	REGION D1.6.1
	    //D1.6.1
	    #"D1.6.1"(ConveyorID := _."D1.6.1",
	              ConveyorSensor:=_."ASiGW-MCC001-bw200-C1: Input"."Sensor D1.6.1",
	              Fault := DB_UDI.ProductionLine.Fault.Stop.Conveyor[_."D1.6.1"],
	              Upstream := DB_UDI.ProductionLine.Upstream.Conveyor[_."D1.6.1"],
	              Downstream := DB_UDI.ProductionLine.DownstreamAccu.Stop.Conveyor[_."D1.6.1"],
	              Interlock := DB_UDI.ProductionLine.Interlock.Stop.Conveyor[_."D1.6.1"],
	              RunForward=>_."ASiGW-MCC001-bw200-C1: Output"."Motor D1.6.1",
	              WriteAsiDir=>_."ASiGW-MCC001-bw200-C1: Output"."Dir D1.6.1");
	    
	END_REGION
	
	REGION D1.7.1
	    //D1.7.1
	    #"D1.7.1"(ConveyorID := _."D1.7.1",
	              ConveyorSensor:=_."ASiGW-MCC001-bw200-C1: Input"."Sensor D1.7.10",
	              Fault := DB_UDI.ProductionLine.Fault.Stop.Conveyor[_."D1.7.1"],
	              Upstream := DB_UDI.ProductionLine.Upstream.Conveyor[_."D1.7.1"],
	              Downstream := DB_UDI.ProductionLine.DownstreamAccu.Stop.Conveyor[_."D1.7.1"],
	              Interlock := DB_UDI.ProductionLine.Interlock.Stop.Conveyor[_."D1.7.1"],
	              RunForward=>_."ASiGW-MCC001-bw200-C1: Output"."Motor D1.7.1",
	              WriteAsiDir=>_."ASiGW-MCC001-bw200-C1: Output"."Dir D1.7.1");
	    
	END_REGION
	
	REGION D1.7.2
	    //D1.7.2
	    #"D1.7.2"(ConveyorID := _."D1.7.2",
	              ConveyorSensor:=_."ASiGW-MCC001-bw200-C1: Input"."Sensor D1.7.10",
	              Fault := DB_UDI.ProductionLine.Fault.Stop.Conveyor[_."D1.7.2"],
	              Upstream := DB_UDI.ProductionLine.Upstream.Conveyor[_."D1.7.2"],
	              Downstream := DB_UDI.ProductionLine.DownstreamAccu.Stop.Conveyor[_."D1.7.2"],
	              Interlock := DB_UDI.ProductionLine.Interlock.Stop.Conveyor[_."D1.7.2"],
	              RunForward=>_."ASiGW-MCC001-bw200-C1: Output"."Motor D1.7.2",
	              WriteAsiDir=>_."ASiGW-MCC001-bw200-C1: Output"."Dir D1.7.2");
	    
	END_REGION
	
	REGION D1.7.3
	    //D1.7.3
	    #"D1.7.3"(ConveyorID := _."D1.7.3",
	              ConveyorSensor:=_."ASiGW-MCC001-bw200-C1: Input"."Sensor D1.7.10",
	              Fault := DB_UDI.ProductionLine.Fault.Stop.Conveyor[_."D1.7.3"],
	              Upstream := DB_UDI.ProductionLine.Upstream.Conveyor[_."D1.7.3"],
	              Downstream := DB_UDI.ProductionLine.DownstreamAccu.Stop.Conveyor[_."D1.7.3"],
	              Interlock := DB_UDI.ProductionLine.Interlock.Stop.Conveyor[_."D1.7.3"],
	              RunForward=>_."ASiGW-MCC001-bw200-C1: Output"."Motor D1.7.3",
	              WriteAsiDir=>_."ASiGW-MCC001-bw200-C1: Output"."Dir D1.7.3");
	    
	END_REGION
	
	REGION D1.7.4
	    //D1.7.4
	    #"D1.7.4"(ConveyorID := _."D1.7.4",
	              ConveyorSensor:=_."ASiGW-MCC001-bw200-C1: Input"."Sensor D1.7.10",
	              Fault := DB_UDI.ProductionLine.Fault.Stop.Conveyor[_."D1.7.4"],
	              Upstream := DB_UDI.ProductionLine.Upstream.Conveyor[_."D1.7.4"],
	              Downstream := DB_UDI.ProductionLine.DownstreamAccu.Stop.Conveyor[_."D1.7.4"],
	              Interlock := DB_UDI.ProductionLine.Interlock.Stop.Conveyor[_."D1.7.4"],
	              RunForward=>_."ASiGW-MCC001-bw200-C1: Output"."Motor D1.7.4",
	              WriteAsiDir=>_."ASiGW-MCC001-bw200-C1: Output"."Dir D1.7.4");
	    
	END_REGION
	
	REGION D1.7.5
	    //D1.7.5
	    #"D1.7.5"(ConveyorID := _."D1.7.5",
	              ConveyorSensor:=_."ASiGW-MCC001-bw200-C1: Input"."Sensor D1.7.10",
	              Fault := DB_UDI.ProductionLine.Fault.Stop.Conveyor[_."D1.7.5"],
	              Upstream := DB_UDI.ProductionLine.Upstream.Conveyor[_."D1.7.5"],
	              Downstream := DB_UDI.ProductionLine.DownstreamAccu.Stop.Conveyor[_."D1.7.5"],
	              Interlock := DB_UDI.ProductionLine.Interlock.Stop.Conveyor[_."D1.7.5"],
	              RunForward=>_."ASiGW-MCC001-bw200-C1: Output"."Motor D1.7.5",
	              WriteAsiDir=>_."ASiGW-MCC001-bw200-C1: Output"."Dir D1.7.5");
	    
	END_REGION
	
	REGION D1.7.6
	    //D1.7.6
	    #"D1.7.6"(ConveyorID := _."D1.7.6",
	              ConveyorSensor:=_."ASiGW-MCC001-bw200-C1: Input"."Sensor D1.7.10",
	              Fault := DB_UDI.ProductionLine.Fault.Stop.Conveyor[_."D1.7.6"],
	              Upstream := DB_UDI.ProductionLine.Upstream.Conveyor[_."D1.7.6"],
	              Downstream := DB_UDI.ProductionLine.DownstreamAccu.Stop.Conveyor[_."D1.7.6"],
	              Interlock := DB_UDI.ProductionLine.Interlock.Stop.Conveyor[_."D1.7.6"],
	              RunForward=>_."ASiGW-MCC001-bw200-C1: Output"."Motor D1.7.6",
	              WriteAsiDir=>_."ASiGW-MCC001-bw200-C1: Output"."Dir D1.7.6");
	    
	END_REGION
	
	REGION D1.7.7
	    //D1.7.7
	    #"D1.7.7"(ConveyorID := _."D1.7.7",
	              ConveyorSensor:=_."ASiGW-MCC001-bw200-C1: Input"."Sensor D1.7.10",
	              Fault := DB_UDI.ProductionLine.Fault.Stop.Conveyor[_."D1.7.7"],
	              Upstream := DB_UDI.ProductionLine.Upstream.Conveyor[_."D1.7.7"],
	              Downstream := DB_UDI.ProductionLine.DownstreamAccu.Stop.Conveyor[_."D1.7.7"],
	              Interlock := DB_UDI.ProductionLine.Interlock.Stop.Conveyor[_."D1.7.7"],
	              RunForward => _."ASiGW-MCC001-bw200-C1: Output"."Motor D1.7.7",
	              WriteAsiDir => _."ASiGW-MCC001-bw200-C1: Output"."Dir D1.7.7");
	    
	END_REGION
	
	REGION D1.7.8
	    //D1.7.8
	    #"D1.7.8"(ConveyorID := _."D1.7.8",
	              ConveyorSensor:=_."ASiGW-MCC001-bw200-C1: Input"."Sensor D1.7.10",
	              Fault := DB_UDI.ProductionLine.Fault.Stop.Conveyor[_."D1.7.8"],
	              Upstream := DB_UDI.ProductionLine.Upstream.Conveyor[_."D1.7.8"],
	              Downstream := DB_UDI.ProductionLine.DownstreamAccu.Stop.Conveyor[_."D1.7.8"],
	              Interlock := DB_UDI.ProductionLine.Interlock.Stop.Conveyor[_."D1.7.8"],
	              RunForward=>_."ASiGW-MCC001-bw200-C1: Output"."Motor D1.7.8",
	              WriteAsiDir=>_."ASiGW-MCC001-bw200-C1: Output"."Dir D1.7.8");
	    
	END_REGION
	
	REGION D1.7.9
	    //D1.7.9
	    #"D1.7.9"(ConveyorID := _."D1.7.9",
	              ConveyorSensor:=_."ASiGW-MCC001-bw200-C1: Input"."Sensor D1.7.10",
	               Fault := DB_UDI.ProductionLine.Fault.Stop.Conveyor[_."D1.7.9"],
	               Upstream := DB_UDI.ProductionLine.Upstream.Conveyor[_."D1.7.9"],
	               Downstream := DB_UDI.ProductionLine.DownstreamAccu.Stop.Conveyor[_."D1.7.9"],
	               Interlock := DB_UDI.ProductionLine.Interlock.Stop.Conveyor[_."D1.7.9"],
	               RunForward=>_."ASiGW-MCC001-bw200-C1: Output"."Motor D1.7.9",
	               WriteAsiDir=>_."ASiGW-MCC001-bw200-C1: Output"."Dir D1.7.9");
	     
	END_REGION
	
	REGION D1.7.10
	    //D1.7.10
	    #"D1.7.10"(ConveyorID := _."D1.7.10",
	               ConveyorSensor:=_."ASiGW-MCC001-bw200-C1: Input"."Sensor D1.7.10",
	               Fault := DB_UDI.ProductionLine.Fault.Stop.Conveyor[_."D1.7.10"],
	               Upstream := DB_UDI.ProductionLine.Upstream.Conveyor[_."D1.7.10"],
	               Downstream := DB_UDI.ProductionLine.DownstreamAccu.Stop.Conveyor[_."D1.7.10"],
	               Interlock := DB_UDI.ProductionLine.Interlock.Stop.Conveyor[_."D1.7.10"],
	               RunForward => _."ASiGW-MCC001-bw200-C1: Output"."Motor D1.7.10",
	               WriteAsiDir => _."ASiGW-MCC001-bw200-C1: Output"."Dir D1.7.10");
	    
	END_REGION
	
	REGION D1.8.1
	    //D1.8.1
	    #"D1.8.1"(ConveyorID := _."D1.8.1",
	              ConveyorSensor:=_."ASiGW-MCC001-bw200-C1: Input"."Sensor D1.8.1",
	              Fault := DB_UDI.ProductionLine.Fault.Stop.Conveyor[_."D1.8.1"],
	              Upstream := DB_UDI.ProductionLine.Upstream.Conveyor[_."D1.8.1"],
	              Downstream := DB_UDI.ProductionLine.DownstreamAccu.Stop.Conveyor[_."D1.8.1"],
	              Interlock := DB_UDI.ProductionLine.Interlock.Stop.Conveyor[_."D1.8.1"],
	              RunForward => _."ASiGW-MCC001-bw200-C1: Output"."Motor D1.8.1",
	              WriteAsiDir => _."ASiGW-MCC001-bw200-C1: Output"."Dir D1.8.1");
	    
	END_REGION
	
	REGION D1.8.2
	    //D1.8.2
	    #"D1.8.2"(ConveyorID := _."D1.8.2",
	              ConveyorSensor:=_."ASiGW-MCC001-bw200-C1: Input"."Sensor D1.8.2",
	              Fault := DB_UDI.ProductionLine.Fault.Stop.Conveyor[_."D1.8.2"],
	              Upstream := DB_UDI.ProductionLine.Upstream.Conveyor[_."D1.8.2"],
	              Downstream := DB_UDI.ProductionLine.DownstreamAccu.Stop.Conveyor[_."D1.8.2"],
	              Interlock := DB_UDI.ProductionLine.Interlock.Stop.Conveyor[_."D1.8.2"],
	              RunForward => _."ASiGW-MCC001-bw200-C1: Output"."Motor D1.8.2",
	              WriteAsiDir => _."ASiGW-MCC001-bw200-C1: Output"."Dir D1.8.2");
	    
	END_REGION
	
	REGION D1.8.3
	    //D1.8.3
	    #"D1.8.3"(ConveyorID := _."D1.8.3",
	              ConveyorSensor:=_."ASiGW-MCC001-bw200-C1: Input"."Sensor D1.8.3",
	              Fault := DB_UDI.ProductionLine.Fault.Stop.Conveyor[_."D1.8.3"],
	              Upstream := DB_UDI.ProductionLine.Upstream.Conveyor[_."D1.8.3"],
	              Downstream := DB_UDI.ProductionLine.DownstreamAccu.Stop.Conveyor[_."D1.8.3"],
	              Interlock := DB_UDI.ProductionLine.Interlock.Stop.Conveyor[_."D1.8.3"],
	              RunForward => _."ASiGW-MCC001-bw200-C1: Output"."Motor D1.8.3",
	              WriteAsiDir => _."ASiGW-MCC001-bw200-C1: Output"."Dir D1.8.3");
	    
	END_REGION
	
	REGION D1.9.1 Transfer Unit
	    ////Transfer D1.9.1
	    #"D1.9.2"(TransferID := _."D1.9.1",
	              TransferSensor:=_."ASiGW-MCC001-bw200-C1: Input"."LoadPresence -D1.9.1",
	              Fault := DB_UDI.ProductionLine.Fault.Stop.Conveyor[_."D1.9.1"],
	              Upstream := DB_UDI.ProductionLine.Upstream.Conveyor[_."D1.9.1"],
	              FrontSensor:=_."ASiGW-MCC001-bw200-C1: Input"."FrontSensor -D1.9.1",
	              EndSensor:=_."ASiGW-MCC001-bw200-C1: Input"."EndSensor -D1.9.1",
	              "Left/RightSensor":=_."ASiGW-MCC001-bw200-C1: Input"."LeftSensor -D1.9.1",
	              Downstream := DB_UDI.ProductionLine.DownstreamAccu.Stop.Conveyor[_."D1.9.1"],
	              TransferDirection := DB_ToteTracking.Conveyor[_."D1.9.1"].ToteDir,
	              StartSignal => _."ASiGW-MCC001-bw200-C1: Output"."StartSignal -D1.9.1",
	              Cmd1 =>  _."ASiGW-MCC001-bw200-C1: Output"."Command1 -D1.9.1",
	              Cmd2 => _."ASiGW-MCC001-bw200-C1: Output"."Command2 -D1.9.1",
	              ErrorReset =>  _."ASiGW-MCC001-bw200-C1: Output"."ErrorReset -D1.9.1");
	    
	END_REGION
	
	REGION D1.10.1 Transfer Unit
	    ////Transfer D1.10.1
	    #"D1.10.1"(TransferID := _."D1.10.1",
	              Fault := DB_UDI.ProductionLine.Fault.Stop.Conveyor[_."D1.10.1"],
	              Upstream := DB_UDI.ProductionLine.Upstream.Conveyor[_."D1.10.1"],
	              Downstream := DB_UDI.ProductionLine.DownstreamAccu.Stop.Conveyor[_."D1.10.1"],
	              TransferDirection := DB_ToteTracking.Conveyor[_."D1.10.1"].ToteDir,
	              StartSignal =>  _."ASiGW-MCC001-bw200-C1: Output"."StartSignal -D1.10.1",
	              Cmd1 =>  _."ASiGW-MCC001-bw200-C1: Output"."Command1 -D1.10.1",
	              Cmd2 =>  _."ASiGW-MCC001-bw200-C1: Output"."Command2 -D1.10.1",
	              ErrorReset =>  _."ASiGW-MCC001-bw200-C1: Output"."ErrorReset -D1.10.1");
	    
	END_REGION
	
	REGION D1.11.1
	    //D1.11.1
	    #"D1.11.1"(ConveyorID := _."D1.11.1",
	               ConveyorSensor:=_."ASiGW-MCC001-bw200-C1: Input"."Sensor D1.11.1",
	               Fault := DB_UDI.ProductionLine.Fault.Stop.Conveyor[_."D1.11.1"],
	               Upstream := DB_UDI.ProductionLine.Upstream.Conveyor[_."D1.11.1"],
	               Downstream := DB_UDI.ProductionLine.DownstreamAccu.Stop.Conveyor[_."D1.11.1"],
	               Interlock := DB_UDI.ProductionLine.Interlock.Stop.Conveyor[_."D1.11.1"],
	               RunForward => _."ASiGW-MCC001-bw200-C1: Output"."Motor D1.11.1",
	               WriteAsiDir => _."ASiGW-MCC001-bw200-C1: Output"."Dir D1.11.1");
	    
	END_REGION
	
	REGION D1.11.2
	    //D1.11.2
	    #"D1.11.2"(ConveyorID := _."D1.11.2",
	               ConveyorSensor:=_."ASiGW-MCC001-bw200-C1: Input"."Sensor D1.11.2",
	               Fault := DB_UDI.ProductionLine.Fault.Stop.Conveyor[_."D1.11.2"],
	               Upstream := DB_UDI.ProductionLine.Upstream.Conveyor[_."D1.11.2"],
	               Downstream := DB_UDI.ProductionLine.DownstreamAccu.Stop.Conveyor[_."D1.11.2"],
	               Interlock := DB_UDI.ProductionLine.Interlock.Stop.Conveyor[_."D1.11.2"],
	               RunForward => _."ASiGW-MCC001-bw200-C1: Output"."Motor D1.11.2",
	               WriteAsiDir => _."ASiGW-MCC001-bw200-C1: Output"."Dir D1.11.2");
	    
	END_REGION
	
	REGION D1.11.3
	    //D1.11.3
	    #"D1.11.3"(ConveyorID := _."D1.11.3",
	               ConveyorSensor:=_."ASiGW-MCC001-bw200-C1: Input"."Sensor D1.11.3",
	               Fault := DB_UDI.ProductionLine.Fault.Stop.Conveyor[_."D1.11.3"],
	               Upstream := DB_UDI.ProductionLine.Upstream.Conveyor[_."D1.11.3"],
	               Downstream := DB_UDI.ProductionLine.DownstreamAccu.Stop.Conveyor[_."D1.11.3"],
	               Interlock := DB_UDI.ProductionLine.Interlock.Stop.Conveyor[_."D1.11.3"],
	               RunForward => _."ASiGW-MCC001-bw200-C1: Output"."Motor D1.11.3",
	               WriteAsiDir => _."ASiGW-MCC001-bw200-C1: Output"."Dir D1.11.3");
	    
	END_REGION
	
	REGION D1.12.1
	    //D1.12.1
	    #"D1.12.1"(ConveyorID := _."D1.12.1",
	               ConveyorSensor:=_."ASiGW-MCC001-bw200-C1: Input"."Sensor D1.12.3",
	               Fault := DB_UDI.ProductionLine.Fault.Stop.Conveyor[_."D1.12.1"],
	               Upstream := DB_UDI.ProductionLine.Upstream.Conveyor[_."D1.12.1"],
	               Downstream := DB_UDI.ProductionLine.DownstreamAccu.Stop.Conveyor[_."D1.12.1"],
	               Interlock := DB_UDI.ProductionLine.Interlock.Stop.Conveyor[_."D1.12.1"],
	               RunForward=>_."ASiGW-MCC001-bw200-C1: Output"."Motor D1.12.1",
	               WriteAsiDir=>_."ASiGW-MCC001-bw200-C1: Output"."Dir D1.12.1");
	    
	END_REGION
	
	REGION D1.12.2
	    //D1.12.2
	    #"D1.12.2"(ConveyorID := _."D1.12.2",
	               ConveyorSensor:=_."ASiGW-MCC001-bw200-C1: Input"."Sensor D1.12.3",
	               Fault := DB_UDI.ProductionLine.Fault.Stop.Conveyor[_."D1.12.2"],
	               Upstream := DB_UDI.ProductionLine.Upstream.Conveyor[_."D1.12.2"],
	               Downstream := DB_UDI.ProductionLine.DownstreamAccu.Stop.Conveyor[_."D1.12.2"],
	               Interlock := DB_UDI.ProductionLine.Interlock.Stop.Conveyor[_."D1.12.2"],
	               RunForward => _."ASiGW-MCC001-bw200-C1: Output"."Motor D1.12.2",
	               WriteAsiDir => _."ASiGW-MCC001-bw200-C1: Output"."Dir D1.12.2");
	    
	END_REGION
	
	REGION D1.12.3
	    ////End
	    #"D1.12.3"(ConveyorID := _."D1.12.3",
	               ConveyorSensor:=_."ASiGW-MCC001-bw200-C1: Input"."Sensor D1.12.3",
	               Fault := DB_UDI.ProductionLine.Fault.Stop.Conveyor[_."D1.12.3"],
	               Upstream := DB_UDI.ProductionLine.Upstream.Conveyor[_."D1.12.3"],
	               Downstream := DB_UDI.ProductionLine.DownstreamAccu.Stop.Conveyor[_."D1.12.3"],
	               Interlock := DB_UDI.ProductionLine.Interlock.Stop.Conveyor[_."D1.12.3"],
	               RunForward => _."ASiGW-MCC001-bw200-C1: Output"."Motor D1.12.3",
	               WriteAsiDir => _."ASiGW-MCC001-bw200-C1: Output"."Dir D1.12.3");
	    
	END_REGION
	
	REGION E1.1.1
	    //E1.1.1
	    #"E1.1.1"(ConveyorID := _."E1.1.1",
	              ConveyorSensor:=_."ASiGW-MCC001-bw200-C1: Input"."Sensor E1.1.1",
	              Fault := DB_UDI.ProductionLine.Fault.Stop.Conveyor[_."E1.1.1"],
	              Upstream := DB_UDI.ProductionLine.Upstream.Conveyor[_."E1.1.1"],
	              Downstream := DB_UDI.ProductionLine.DownstreamAccu.Stop.Conveyor[_."E1.1.1"],
	              Interlock := DB_UDI.ProductionLine.Interlock.Stop.Conveyor[_."E1.1.1"],
	              RunForward=>_."ASiGW-MCC001-bw200-C1: Output"."Motor E1.1.1",
	              WriteAsiDir=>_."ASiGW-MCC001-bw200-C1: Output"."Dir E1.1.1");
	    
	END_REGION
	
	REGION E1.1.2
	    //E1.1.2
	    #"E1.1.2"(ConveyorID := _."E1.1.2",
	              ConveyorSensor:=_."ASiGW-MCC001-bw200-C1: Input"."Sensor E1.1.4",
	              Fault := DB_UDI.ProductionLine.Fault.Stop.Conveyor[_."E1.1.2"],
	              Upstream := DB_UDI.ProductionLine.Upstream.Conveyor[_."E1.1.2"],
	              Downstream := DB_UDI.ProductionLine.DownstreamAccu.Stop.Conveyor[_."E1.1.2"],
	              Interlock := DB_UDI.ProductionLine.Interlock.Stop.Conveyor[_."E1.1.2"],
	              RunForward=>_."ASiGW-MCC001-bw200-C1: Output"."Motor E1.1.2",
	              WriteAsiDir=>_."ASiGW-MCC001-bw200-C1: Output"."Dir E1.1.2");
	    
	END_REGION
	
	REGION E1.1.3
	    //E1.1.3
	    #"E1.1.3"(ConveyorID := _."E1.1.3",
	              ConveyorSensor:=_."ASiGW-MCC001-bw200-C1: Input"."Sensor E1.1.4",
	              Fault := DB_UDI.ProductionLine.Fault.Stop.Conveyor[_."E1.1.3"],
	              Upstream := DB_UDI.ProductionLine.Upstream.Conveyor[_."E1.1.3"],
	              Downstream := DB_UDI.ProductionLine.DownstreamAccu.Stop.Conveyor[_."E1.1.3"],
	              Interlock := DB_UDI.ProductionLine.Interlock.Stop.Conveyor[_."E1.1.3"],
	              RunForward=>_."ASiGW-MCC001-bw200-C1: Output"."Motor E1.1.3",
	              WriteAsiDir=>_."ASiGW-MCC001-bw200-C1: Output"."Dir E1.1.3");
	    
	END_REGION
	
	REGION E1.1.4
	    //E1.1.4
	    #"E1.1.4"(ConveyorID := _."E1.1.4",
	              ConveyorSensor:=_."ASiGW-MCC001-bw200-C1: Input"."Sensor E1.1.4",
	              Fault := DB_UDI.ProductionLine.Fault.Stop.Conveyor[_."E1.1.4"],
	              Upstream := DB_UDI.ProductionLine.Upstream.Conveyor[_."E1.1.4"],
	              Downstream := DB_UDI.ProductionLine.DownstreamAccu.Stop.Conveyor[_."E1.1.4"],
	              Interlock := DB_UDI.ProductionLine.Interlock.Stop.Conveyor[_."E1.1.4"],
	              RunForward=>_."ASiGW-MCC001-bw200-C1: Output"."Motor E1.1.4",
	              WriteAsiDir=>_."ASiGW-MCC001-bw200-C1: Output"."Dir E1.1.4");
	    
	END_REGION
	
	REGION E1.2.1
	    //E1.2.1
	    #"E1.2.1"(ConveyorID := _."E1.2.1",
	              ConveyorSensor:=_."ASiGW-MCC001-bw200-C1: Input"."Sensor E1.2.1",
	              Fault := DB_UDI.ProductionLine.Fault.Stop.Conveyor[_."E1.2.1"],
	              Upstream := DB_UDI.ProductionLine.Upstream.Conveyor[_."E1.2.1"],
	              Downstream := DB_UDI.ProductionLine.DownstreamAccu.Stop.Conveyor[_."E1.2.1"],
	              Interlock := DB_UDI.ProductionLine.Interlock.Stop.Conveyor[_."E1.2.1"],
	              RunForward=>_."ASiGW-MCC001-bw200-C1: Output"."Motor - E1.2.1",
	              WriteAsiDir=>_."ASiGW-MCC001-bw200-C1: Output"."1-21A Dir",
	              WriteAsiSpeed=>_."ASiGW-MCC001-bw200-C1: Output"."1-21A Speed");
	    
	END_REGION
	
	REGION E1.3.1
	    //E1.3.1
	    #"E1.3.1"(ConveyorID := _."E1.3.1",
	              ConveyorSensor:=_."ASiGW-MCC001-bw200-C1: Input"."Sensor E1.3.1",
	              Fault := DB_UDI.ProductionLine.Fault.Stop.Conveyor[_."E1.3.1"],
	              Upstream := DB_UDI.ProductionLine.Upstream.Conveyor[_."E1.3.1"],
	              Downstream := DB_UDI.ProductionLine.DownstreamAccu.Stop.Conveyor[_."E1.3.1"],
	              Interlock := DB_UDI.ProductionLine.Interlock.Stop.Conveyor[_."E1.3.1"],
	              RunForward=>_."ASiGW-MCC001-bw200-C1: Output"."Motor - E1.3.1",
	              WriteAsiDir=>_."ASiGW-MCC001-bw200-C1: Output"."1-21A Dir",
	              WriteAsiSpeed=>_."ASiGW-MCC001-bw200-C1: Output"."1-21A Speed");
	    
	END_REGION
	
	REGION E1.4.1
	    //E1.4.1
	    #"E1.4.1"(ConveyorID := _."E1.4.1",
	              ConveyorSensor:=_."ASiGW-MCC001-bw200-C1: Input"."Sensor E1.4.1",
	              Fault := DB_UDI.ProductionLine.Fault.Stop.Conveyor[_."E1.4.1"],
	              Upstream := DB_UDI.ProductionLine.Upstream.Conveyor[_."E1.4.1"],
	              Downstream := DB_UDI.ProductionLine.DownstreamAccu.Stop.Conveyor[_."E1.4.1"],
	              Interlock := DB_UDI.ProductionLine.Interlock.Stop.Conveyor[_."E1.4.1"],
	              RunForward=>_."ASiGW-MCC001-bw200-C1: Output"."Motor E1.4.1",
	              WriteAsiDir=>_."ASiGW-MCC001-bw200-C1: Output"."Dir E1.4.1");
	    
	END_REGION
	
	REGION E1.5.1
	    //E1.5.1
	    #"E1.5.1"(ConveyorID := _."E1.5.1",
	              ConveyorSensor := _."ASiGW-MCC001-bw200-C1: Input"."Sensor E1.5.1",
	              Fault := DB_UDI.ProductionLine.Fault.Stop.Conveyor[_."E1.5.1"],
	              Upstream := DB_UDI.ProductionLine.Upstream.Conveyor[_."E1.5.1"],
	              Downstream := DB_UDI.ProductionLine.DownstreamAccu.Stop.Conveyor[_."E1.5.1"],
	              Interlock := DB_UDI.ProductionLine.Interlock.Stop.Conveyor[_."E1.5.1"],
	              RunForward => _."ASiGW-MCC001-bw200-C1: Output"."Motor - E1.5.1",
	              WriteAsiDir => _."ASiGW-MCC001-bw200-C1: Output"."1-23A Dir",
	              WriteAsiSpeed => _."ASiGW-MCC001-bw200-C1: Output"."1-23A Speed");
	    
	    
	END_REGION
	
	REGION E1.6.1
	    ////E1.6.1 Arm for Merger2
	    #"E1.6.1"(ConveyorID := _."E1.6.1",
	              ConveyorSensor:=_."ASiGW-MCC001-bw200-C1: Input"."Sensor E1.5.1",
	              Fault := DB_UDI.ProductionLine.Fault.Stop.Conveyor[_."E1.6.1"],
	              Upstream := DB_UDI.ProductionLine.Upstream.Conveyor[_."E1.6.1"],
	              Downstream := DB_UDI.ProductionLine.DownstreamAccu.Stop.Conveyor[_."E1.6.1"],
	              Interlock := DB_UDI.ProductionLine.Interlock.Stop.Conveyor[_."E1.6.1"],
	              RunForward=>_."ASiGW-MCC001-bw200-C1: Output"."Motor E1.6.1",
	              WriteAsiDir=>_."ASiGW-MCC001-bw200-C1: Output"."Dir E1.6.1");
	    
	END_REGION
	
	
END_FUNCTION_BLOCK
END_NAMESPACE

NAMESPACE ProductionLine
ORGANIZATION_BLOCK Main_ProductionLine
TITLE = "Main Program Sweep (Cycle)"
{ S7_Optimized_Access := 'TRUE' ; Published := 'FALSE' }
VERSION : 0.1

BEGIN
	// ==========================================================================================================================================
	// Company        : LogTech, s.r.o.
	// Created by     : Mahmoud Elnady
	// Block          : FB_Main_ProductionLine
	// Project        : Lékárna Chrudim
	// Project number : 23-157
	// ==========================================================================================================================================
	
	//Synchronization Line_A1 and Global
	
	REGION Synchronization
	    
	    FC_Sync();
	    
	END_REGION
	
	REGION Line A1
	    
	    IDB_ProductionLine();
	    
	    //Upstream
	    FC_Upstream();
	    
	    //Downstream
	    FC_Downstream();
	    
	    //Fault
	    FC_Fault();
	    
	    // Merging
	    IDB_Merging();
	    
	    // Barcode
	    IDB_BarcodeReader();
	    
	    // OPC Server
	    IDB_OPC_Communication();
	    
	    //FB Technology
	    IDB_FB_Technology();
	    
	    //Tote Tracking
	    IDB_ToteTracking();
	    
	    // FB Segments Status
	    IDB_Segments_Status();
	    
	    // FB Toggle Dir
	    IDB_FB_ToggleDir();
	    
	    //FC Alarm
	    FC_Alarm();
	    
	END_REGION
	
	REGION Test
	    // Flow Test
	    IDB_Flow_Test();
	    
	END_REGION
	
	
	
	
	
	
	
	
	
	
	
	
END_ORGANIZATION_BLOCK
END_NAMESPACE

NAMESPACE Global
FUNCTION FC_ReadSystemSSR : Void
{ S7_Optimized_Access := 'TRUE' ; Published := 'FALSE' }
VERSION : 0.1

BEGIN
	// ==========================================================================================================================================
	// Company        : LogTech, s.r.o.
	// Created by     : Anton Vinoth Soundraraj
	// Block          : FC_ReadSystemSSR
	// Project        : Lékarna DC Chrudim
	// Project number : 23-157
	// ==========================================================================================================================================
	
	REGION Line A1
	    
	    // Start Stop Reset IO
	    
	    // Activate Start bit
	    DB_SystemSSR.Line.A1.StartSystem :=
	    DB_SystemSSR.FromHMI.Line.A1.StartSystem;
	    // Activate Stop bit
	    DB_SystemSSR.Line.A1.StopSystem :=
	    DB_SystemSSR.FromHMI.Line.A1.StopSystem;
	    // Activate Reset bit
	    DB_SystemSSR.Line.A1.ResetSystem :=
	    DB_SystemSSR.FromHMI.Line.A1.ResetSystem;
	    
	END_REGION
	
	REGION Line B1
	    
	    // Start Stop Reset IO
	    
	    // Activate Start bit
	    DB_SystemSSR.Line.B1.StartSystem :=
	    DB_SystemSSR.FromHMI.Line.B1.StartSystem;
	    // Activate Stop bit
	    DB_SystemSSR.Line.B1.StopSystem :=
	    DB_SystemSSR.FromHMI.Line.B1.StopSystem;
	    // Activate Reset bit
	    DB_SystemSSR.Line.B1.ResetSystem :=
	    DB_SystemSSR.FromHMI.Line.B1.ResetSystem;
	    
	END_REGION
	
	REGION Line C1
	    
	    // Start Stop Reset IO
	    
	    // Activate Start bit
	    DB_SystemSSR.Line.C1.StartSystem :=
	    DB_SystemSSR.FromHMI.Line.C1.StartSystem OR
	    _.DB_Sync.startbit;
	    // Activate Stop bit
	    DB_SystemSSR.Line.C1.StopSystem :=
	    DB_SystemSSR.FromHMI.Line.C1.StopSystem OR
	    _.DB_Sync.stopbit;
	    // Activate Reset bit
	    DB_SystemSSR.Line.C1.ResetSystem :=
	    DB_SystemSSR.FromHMI.Line.C1.ResetSystem OR
	    _.DB_Sync.resetbit;
	    
	END_REGION
	
	REGION Line D1
	    
	    // Start Stop Reset IO
	    
	    // Activate Start bit
	    DB_SystemSSR.Line.D1.StartSystem :=
	    DB_SystemSSR.FromHMI.Line.D1.StartSystem;
	    // Activate Stop bit
	    DB_SystemSSR.Line.D1.StopSystem :=
	    DB_SystemSSR.FromHMI.Line.D1.StopSystem;
	    // Activate Reset bit
	    DB_SystemSSR.Line.D1.ResetSystem :=
	    DB_SystemSSR.FromHMI.Line.D1.ResetSystem;
	    
	END_REGION
END_FUNCTION
END_NAMESPACE

NAMESPACE Global
FUNCTION_BLOCK FB_Conveyor
{ S7_Optimized_Access := 'TRUE' ; Published := 'TRUE' }
VERSION : 0.1
   VAR_INPUT 
      ConveyorID : Int;
      ConveyorSensor : Bool;
      Fault : Bool;
      Upstream : Bool;
      Downstream : Bool;
      Interlock : Bool;
   END_VAR

   VAR_OUTPUT 
      RunForward : Bool;
      WriteAsiDir : Bool;
      WriteAsiSpeed : Bool;
      NordControlEnable : Word;
      NordSetpoint : Word;
   END_VAR

   VAR 
      sConvID : Int;
      ReadInputSignal : Struct
         ConveyorSensor : Bool;
         EmergencyStop : Bool;
         Fault : Bool;
      END_STRUCT;
      MotorType : Struct
         "24v-ASi" : Bool;
         nord : Bool;
      END_STRUCT;
      Active : Struct
         Line : Struct
            A1 : Bool;
            B1 : Bool;
            C1 : Bool;
            D1 : Bool;
         END_STRUCT;
      END_STRUCT;
      CONVEYOR_SENSOR : FB_Sensor;
      CONVEYOR_SENSOR_BLOCKAGE : FB_SensorBlockage;
      CONVEYOR_STATUS_ON : FB_StatusON;
      CONVEYOR_STATUS_READY : FB_StatusReady;
      CONVEYOR_STATUS_FAULT : FB_StatusFault;
      "RUN/STOP_CONVEYOR" : FB_RunStop;
      ENERGY_SAVE : FB_EnergySave;
      AUTO_RESET : FB_AutoReset;
      SSR { S7_SetPoint := 'False'} : SystemSSR;
      ReadConveyorStatus : ConveyorStatus;
      ReadConveyorParameters { S7_SetPoint := 'False'} : ConveyorParameters := ((), [2(T#10ms)], (), (), ());
      ConveyorFault : Fault;
      SimuMode : Struct
         Sensor : Bool;
         Fault : Bool;
         Estop : Struct
            Zone : Struct
               "1" : Bool;
               "2" : Bool;
               "3" : Bool;
               "4" : Bool;
            END_STRUCT;
         END_STRUCT;
      END_STRUCT;
      StartUpTimer {InstructionName := 'TOF_TIME'; LibVersion := '1.0'; S7_SetPoint := 'False'} : TOF_TIME;
      FT_StartUp {InstructionName := 'F_TRIG'; LibVersion := '1.0'} : F_TRIG;
      SetStartUp { S7_SetPoint := 'True'} : Bool;
      FilteredSensor { S7_SetPoint := 'True'} : Bool;
      StopSystemFireActive : Bool;
      EnergySave : Bool;
      StartMotorForward : Bool;
      StartMotorReverse : Bool;
      AutoReset { S7_SetPoint := 'True'} : Bool;
      VisuColor : Word;
      NordSetpointRun : Word := 16#047F;
      NordSetpointReady : Word := 16#047E;
      NordFaultAck : Word := 16#0080;
   END_VAR


BEGIN
	// ==========================================================================================================================================
	// Company        : LogTech, s.r.o.
	// Created by     : Anton Vinoth Soundraraj
	// Block          : FB_Conveyor
	// Project        : Lékarna DC Chrudim
	// Project number : 23-157
	// ==========================================================================================================================================
	
	// input to static
	#sConvID := #ConveyorID;
	
	REGION Active Line
	    
	    // Line A1
	    IF (#ConveyorID >= _.gMinA1 AND
	        #ConveyorID <= _.gMaxA1)
	    THEN
	        #Active.Line.A1 := TRUE;
	    END_IF;
	    
	    // Line B1
	    IF (#ConveyorID >= _.gMinB1 AND
	        #ConveyorID <= _.gMaxB1)
	    THEN
	        #Active.Line.B1 := TRUE;
	    END_IF;
	    
	    // Line C1
	    IF (#ConveyorID >= _.gMinC1 AND
	        #ConveyorID <= _.gMaxC1)
	    THEN
	        #Active.Line.C1 := TRUE;
	    END_IF;
	    
	    // Line D1
	    IF (#ConveyorID >= _.gMinD1 AND
	        #ConveyorID <= _.gMaxD1)
	    THEN
	        #Active.Line.A1 := TRUE;
	    END_IF;
	    
	END_REGION 
	
	REGION SystemSSR
	    
	    // Line A1
	    IF #Active.Line.A1 THEN
	        #SSR.StartSystem := DB_SystemSSR.Line.A1.StartSystem;
	        #SSR.StopSystem := DB_SystemSSR.Line.A1.StopSystem;
	        #SSR.ResetSystem := DB_SystemSSR.Line.A1.ResetSystem;
	    END_IF;
	    
	    // Line B1
	    IF #Active.Line.B1 THEN
	        #SSR.StartSystem := DB_SystemSSR.Line.B1.StartSystem;
	        #SSR.StopSystem := DB_SystemSSR.Line.B1.StopSystem;
	        #SSR.ResetSystem := DB_SystemSSR.Line.B1.ResetSystem;
	    END_IF;
	    
	    // Line C1
	    IF #Active.Line.C1 THEN
	        #SSR.StartSystem := DB_SystemSSR.Line.C1.StartSystem;
	        #SSR.StopSystem := DB_SystemSSR.Line.C1.StopSystem;
	        #SSR.ResetSystem := DB_SystemSSR.Line.C1.ResetSystem;
	    END_IF;
	    
	    // Line D1
	    IF #Active.Line.D1 THEN
	        #SSR.StartSystem := DB_SystemSSR.Line.D1.StartSystem;
	        #SSR.StopSystem := DB_SystemSSR.Line.D1.StopSystem;
	        #SSR.ResetSystem := DB_SystemSSR.Line.D1.ResetSystem;
	    END_IF;
	    
	END_REGION
	
	REGION Read Simu inputs  
	    
	    // Line A1
	    IF #Active.Line.A1 THEN
	        // read simu
	        #SimuMode.Sensor := DB_SystemSimu.TriggerSensor.Line.A1.Conveyor[#ConveyorID];
	        #SimuMode.Fault := DB_SystemSimu.TriggerFault.Line.A1.Conveyor[#ConveyorID];
	    END_IF;
	    
	    // Line B1
	    IF #Active.Line.B1 THEN
	        // read simu
	        #SimuMode.Sensor := DB_SystemSimu.TriggerSensor.Line.B1.Conveyor[#ConveyorID];
	        #SimuMode.Fault := DB_SystemSimu.TriggerFault.Line.B1.Conveyor[#ConveyorID];
	    END_IF;
	    
	    // Line C1
	    IF #Active.Line.C1 THEN
	        // read simu
	        #SimuMode.Sensor := DB_SystemSimu.TriggerSensor.Line.C1.Conveyor[#ConveyorID];
	        #SimuMode.Fault := DB_SystemSimu.TriggerFault.Line.C1.Conveyor[#ConveyorID];
	    END_IF;
	    
	    // Line D1
	    IF #Active.Line.D1 THEN
	        // read simu
	        #SimuMode.Sensor := DB_SystemSimu.TriggerSensor.Line.D1.Conveyor[#ConveyorID];
	        #SimuMode.Fault := DB_SystemSimu.TriggerFault.Line.D1.Conveyor[#ConveyorID];
	    END_IF;
	    
	END_REGION
	
	REGION Read Input
	    
	    // read all inputs to the block
	    // Conveyor input read signals
	    #ReadInputSignal.ConveyorSensor := #ConveyorSensor OR  ///coment for sim opreation remove NOT
	    #SimuMode.Sensor; // simu call
	    #ReadInputSignal.Fault := #Fault OR
	    #SimuMode.Fault; // simu call;
	    #ReadInputSignal.EmergencyStop := // all estop zones are connected together
	    _.DB_SafetyStandard.ToStandard.EstopActive;
	    
	END_REGION
	
	REGION READ AND INIT
	    
	    REGION Init conveyor parameters
	        
	        // Conveyor Parameter
	        // Line A1
	        IF #Active.Line.A1 THEN
	            #ReadConveyorParameters := DB_ConveyorParameters.Line.A1.Conveyor[#ConveyorID];
	        END_IF;
	        // Line B1
	        IF #Active.Line.B1 THEN
	            #ReadConveyorParameters := DB_ConveyorParameters.Line.B1.Conveyor[#ConveyorID];
	        END_IF;
	        // Line C1
	        IF #Active.Line.C1 THEN
	            #ReadConveyorParameters := DB_ConveyorParameters.Line.C1.Conveyor[#ConveyorID];
	        END_IF;
	        // Line D1
	        IF #Active.Line.D1 THEN
	            #ReadConveyorParameters := DB_ConveyorParameters.Line.D1.Conveyor[#ConveyorID];
	        END_IF;
	        
	    END_REGION
	    
	    REGION Sensor Filter
	        
	        // FB_Sensor
	        // called as MIDB
	        
	        #CONVEYOR_SENSOR(Sensor           := #ReadInputSignal.ConveyorSensor,
	                         SensorFilterTime := #ReadConveyorParameters.SensorFilterTime,
	                         FilteredSensor   => #FilteredSensor);
	        
	    END_REGION
	    
	    REGION FIRE
	        
	        // Fire signal from fire system stops the whole system
	        // System can be reset from Fire status only if the fire signal is deactivated
	        
	        // FIRE ALARM ACTIVE --> STOP SYSTEM
	        IF DB_SystemSimu.Fire THEN
	            #StopSystemFireActive := TRUE;
	        END_IF;
	        // RESET --> FIRE ALARM
	        IF #SSR.ResetSystem AND NOT DB_SystemSimu.Fire THEN
	            #StopSystemFireActive := FALSE;
	        END_IF;
	        
	    END_REGION
	    
	END_REGION
	
	REGION Conveyor startup
	    
	    // Conveyor StartUp: Conveyor startup signal after preset time
	    #StartUpTimer.TOF(IN := #SSR.StartSystem,
	                      PT := #ReadConveyorParameters.StartUpTime);
	    
	    #FT_StartUp(CLK := #StartUpTimer.Q);
	    
	    // set startup after the preset
	    #SetStartUp := #FT_StartUp.Q;
	    
	END_REGION
	
	REGION Conveyor Status
	    
	    REGION Status ON
	        
	        // ----------------------------------------->>>>>>> STATUS ON <<<<<<<-----------------------------------------
	        // FB_ConveyorStatusON
	        // called as IDMB
	        
	        #CONVEYOR_STATUS_ON(SystemStartActive := #SSR.StartSystem,
	                            StatusStop        := #ReadConveyorStatus.Stop,
	                            StatusEStop       := #ReadConveyorStatus.Estop,
	                            StatusManual      := #ReadConveyorStatus.Manual,
	                            StatusFault       := #ReadConveyorStatus.Fault,
	                            FireAlarmActive   := #StopSystemFireActive,
	                            StatusON          => #ReadConveyorStatus.ON);
	        
	    END_REGION
	    
	    REGION Status Ready
	        
	        // ----------------------------------------->>>>>>> STATUS READY <<<<<<<-----------------------------------------
	        // FB_ConveyorStatusReady
	        // called as MIDB
	        
	        #CONVEYOR_STATUS_READY(StatusON        := #ReadConveyorStatus.ON,
	                               StatusESTOP     := #ReadConveyorStatus.Estop,
	                               StatusFAULT     := #ReadConveyorStatus.Fault,
	                               StatusMAN       := #ReadConveyorStatus.Manual,
	                               SignalFIRE      := #StopSystemFireActive,
	                               SystemAlertTime := #ReadConveyorParameters.StartUpTime,
	                               StatusReady     => #ReadConveyorStatus.ReadytoRun);
	        
	    END_REGION
	    
	    REGION Status Occupied
	        
	        // ----------------------------------------->>>>>>> STATUS OCCUPIED <<<<<<<-----------------------------------------
	        #ReadConveyorStatus.Occupied := #FilteredSensor;
	        
	    END_REGION
	    
	    REGION Status Running
	        
	        // ----------------------------------------->>>>>>> STATUS RUNNING <<<<<<<-----------------------------------------
	        
	        #ReadConveyorStatus.Running := #StartMotorForward OR #StartMotorReverse;
	        
	    END_REGION
	    
	    REGION Status Fault
	        
	        // ----------------------------------------->>>>>>> STATUS FAULT <<<<<<<-----------------------------------------
	        
	        // Automatic reset trigger to the needed drive after wakeup from ESTOP power miss (only if needed)
	        // will trigger for every Reset active
	        
	        #AUTO_RESET(AckIN := #SSR.ResetSystem,
	                    Ack   => #AutoReset);
	        
	        // Reading error signal from the motor drive
	        #ConveyorFault.Motor_Error := #ReadInputSignal.Fault;
	        
	        // FC_ConveyorStatusFault
	        #CONVEYOR_STATUS_FAULT(FaultActive   := #ConveyorFault.Motor_Error,
	                               ResetFault    := #SSR.ResetSystem OR #AutoReset,
	                               StatusRunning := #ReadConveyorStatus.Running,
	                               FaultStatus   => #ReadConveyorStatus.Fault);
	        
	    END_REGION
	    
	    REGION Status ESTOP
	        
	        // ----------------------------------------->>>>>>> STATUS ESTOP <<<<<<<-----------------------------------------
	        
	        // EMERGENCY STOP ACTIVE --> STOP SYSTEM
	        IF #ReadInputSignal.EmergencyStop THEN
	            #ReadConveyorStatus.Estop := TRUE;
	        END_IF;
	        // RESET --> EMERGENCY STOP
	        IF #AutoReset AND NOT #ReadInputSignal.EmergencyStop THEN // (reset after 12 seconds) : Auto Reset
	            #ReadConveyorStatus.Estop := FALSE;
	        END_IF;
	        
	    END_REGION
	    
	    REGION Status Manual
	        
	        // ----------------------------------------->>>>>>> STATUS MANUAL <<<<<<<-----------------------------------------
	        
	        // Write to static from IO
	        // ACTIVATE --> MANUAL MODE
	        // Line A1
	        IF #Active.Line.A1 THEN
	            // SET --> MANUAL MODE
	            IF DB_Manual.Line.A1.Conveyor[#ConveyorID].ManualEnable THEN
	                #ReadConveyorStatus.Manual := TRUE;
	            END_IF;
	            // RESET --> MANUAL MODE
	            IF NOT DB_Manual.Line.A1.Conveyor[#ConveyorID].ManualEnable AND #SSR.ResetSystem THEN
	                #ReadConveyorStatus.Manual := FALSE;
	            END_IF;
	        END_IF;
	        // Line B1
	        IF #Active.Line.B1 THEN
	            // SET --> MANUAL MODE
	            IF DB_Manual.Line.B1.Conveyor[#ConveyorID].ManualEnable THEN
	                #ReadConveyorStatus.Manual := TRUE;
	            END_IF;
	            // RESET --> MANUAL MODE
	            IF NOT DB_Manual.Line.B1.Conveyor[#ConveyorID].ManualEnable AND #SSR.ResetSystem THEN
	                #ReadConveyorStatus.Manual := FALSE;
	            END_IF;
	        END_IF;
	        // Line C1
	        IF #Active.Line.C1 THEN
	            // SET --> MANUAL MODE
	            IF DB_Manual.Line.C1.Conveyor[#ConveyorID].ManualEnable THEN
	                #ReadConveyorStatus.Manual := TRUE;
	            END_IF;
	            // RESET --> MANUAL MODE
	            IF NOT DB_Manual.Line.C1.Conveyor[#ConveyorID].ManualEnable AND #SSR.ResetSystem THEN
	                #ReadConveyorStatus.Manual := FALSE;
	            END_IF;
	        END_IF;
	        // Line D1
	        IF #Active.Line.D1 THEN
	            // SET --> MANUAL MODE
	            IF DB_Manual.Line.D1.Conveyor[#ConveyorID].ManualEnable THEN
	                #ReadConveyorStatus.Manual := TRUE;
	            END_IF;
	            // RESET --> MANUAL MODE
	            IF NOT DB_Manual.Line.D1.Conveyor[#ConveyorID].ManualEnable AND #SSR.ResetSystem THEN
	                #ReadConveyorStatus.Manual := FALSE;
	            END_IF;
	        END_IF;
	        
	        // Manual enable and Run from HMI
	        // Line A1
	        IF #Active.Line.A1 THEN
	            IF #ConveyorID = DB_Manual.Conveyor.ID THEN
	                DB_Manual.Line.A1.Conveyor[DB_Manual.Conveyor.ID].ManualEnable := DB_Manual.Conveyor.Enable;
	                DB_Manual.Line.A1.Conveyor[DB_Manual.Conveyor.ID].Run.Forward := DB_Manual.Conveyor.in;
	            END_IF;
	        END_IF;
	        // Line B1
	        IF #Active.Line.B1 THEN
	            IF #ConveyorID = DB_Manual.Conveyor.ID THEN
	                DB_Manual.Line.B1.Conveyor[DB_Manual.Conveyor.ID].ManualEnable := DB_Manual.Conveyor.Enable;
	                DB_Manual.Line.B1.Conveyor[DB_Manual.Conveyor.ID].Run.Forward := DB_Manual.Conveyor.in;
	            END_IF;
	        END_IF;
	        // Line C1
	        IF #Active.Line.C1 THEN
	            IF #ConveyorID = DB_Manual.Conveyor.ID THEN
	                DB_Manual.Line.C1.Conveyor[DB_Manual.Conveyor.ID].ManualEnable := DB_Manual.Conveyor.Enable;
	                DB_Manual.Line.C1.Conveyor[DB_Manual.Conveyor.ID].Run.Forward := DB_Manual.Conveyor.in;
	            END_IF;
	        END_IF;
	        // Line D1
	        IF #Active.Line.D1 THEN
	            IF #ConveyorID = DB_Manual.Conveyor.ID THEN
	                DB_Manual.Line.D1.Conveyor[DB_Manual.Conveyor.ID].ManualEnable := DB_Manual.Conveyor.Enable;
	                DB_Manual.Line.D1.Conveyor[DB_Manual.Conveyor.ID].Run.Forward := DB_Manual.Conveyor.in;
	            END_IF;
	        END_IF;
	        
	    END_REGION
	    
	    REGION Status Stop
	        
	        // ----------------------------------------->>>>>>> STATUS STOP <<<<<<<-----------------------------------------
	        
	        IF #SSR.StopSystem THEN
	            #ReadConveyorStatus.Stop := TRUE;
	        END_IF;
	        IF #SSR.StartSystem OR #SSR.ResetSystem THEN
	            #ReadConveyorStatus.Stop := FALSE;
	        END_IF;
	        
	    END_REGION
	    
	    REGION Sensor Blockage
	        
	        // ----------------------------------------->>>>>>> STATUS BLOCKAGE <<<<<<<------------------------------------
	        
	        // FB_SensorBlockage
	        // called as MIDB
	        #CONVEYOR_SENSOR_BLOCKAGE(ConveyorSensor       := #FilteredSensor,
	                                  StatusRunning        := #ReadConveyorStatus.Running,
	                                  SensorBlockagePeriod := #ReadConveyorParameters.SensorBlockageTime,
	                                  SensorBlocked        => #ConveyorFault.Sensor_Blockage,
	                                  ReadBlockageStatus   => #ReadConveyorStatus.Blockage);
	        
	        REGION alarm 
	            
	            // ==========================
	            // Sensor Blockage: HMI Alarm
	            // ==========================
	            // Sensor blockage alarm message is written to the alarm word
	            // corresponding to the active line
	            // Line A1
	            IF #Active.Line.A1 THEN
	                DB_Alarm."word".Line.A1.Conveyor[#ConveyorID].%X0 := #ReadConveyorStatus.Blockage;
	            END_IF;
	            // Line B1
	            IF #Active.Line.B1 THEN
	                DB_Alarm."word".Line.B1.Conveyor[#ConveyorID].%X0 := #ReadConveyorStatus.Blockage;
	            END_IF;
	            // Line C1
	            IF #Active.Line.C1 THEN
	                DB_Alarm."word".Line.C1.Conveyor[#ConveyorID].%X0 := #ReadConveyorStatus.Blockage;
	            END_IF;
	            // Line D1
	            IF #Active.Line.D1 THEN
	                DB_Alarm."word".Line.D1.Conveyor[#ConveyorID].%X0 := #ReadConveyorStatus.Blockage;
	            END_IF;
	            
	        END_REGION
	        
	    END_REGION
	    
	    REGION Visu Color
	        
	        // each and every status of the conveyor will be mentioned by different colors in HMI panel
	        
	        #VisuColor.%X8 := #ReadConveyorStatus.Blockage;
	        #VisuColor.%X0 := #ReadConveyorStatus.ON;
	        #VisuColor.%X1 := #ReadConveyorStatus.ReadytoRun;
	        #VisuColor.%X2 := #ReadConveyorStatus.Occupied;
	        #VisuColor.%X3 := #ReadConveyorStatus.Running;
	        #VisuColor.%X4 := #ReadConveyorStatus.Fault;
	        #VisuColor.%X5 := #ReadConveyorStatus.Estop;
	        #VisuColor.%X6 := #ReadConveyorStatus.Manual;
	        #VisuColor.%X7 := #ReadConveyorStatus.Stop;
	        
	        // convert word to Interger value: 
	        // color will be depends on the status priority (integer value) 
	        // reference: Conveyor image in HMI screen -> property -> Apperance   
	        
	        // Line A1
	        IF #Active.Line.A1 THEN
	            DB_VisuColor.Line.A1.Conveyor[#ConveyorID] :=
	            WORD_TO_INT(#VisuColor);
	        END_IF;
	        // Line B1
	        IF #Active.Line.B1 THEN
	            DB_VisuColor.Line.B1.Conveyor[#ConveyorID] :=
	            WORD_TO_INT(#VisuColor);
	        END_IF;
	        // Line C1
	        IF #Active.Line.C1 THEN
	            DB_VisuColor.Line.C1.Conveyor[#ConveyorID] :=
	            WORD_TO_INT(#VisuColor);
	        END_IF;
	        // Line D1
	        IF #Active.Line.D1 THEN
	            DB_VisuColor.Line.D1.Conveyor[#ConveyorID] :=
	            WORD_TO_INT(#VisuColor);
	        END_IF;
	        
	    END_REGION
	    
	    REGION Global Status
	        
	        // write -> global status
	        // Line A1
	        IF #Active.Line.A1 THEN
	            DB_Global.Status.Line.A1.On[#ConveyorID] := #ReadConveyorStatus.ON;
	            DB_Global.Status.Line.A1.ReadyToRun[#ConveyorID] := #ReadConveyorStatus.ReadytoRun;
	            DB_Global.Status.Line.A1.Occupied[#ConveyorID] := #ReadConveyorStatus.Occupied;
	            DB_Global.Status.Line.A1.Running[#ConveyorID] := #ReadConveyorStatus.Running;
	            DB_Global.Status.Line.A1.Fault[#ConveyorID] := #ReadConveyorStatus.Fault;
	            DB_Global.Status.Line.A1.Estop[#ConveyorID] := #ReadConveyorStatus.Estop;
	            DB_Global.Status.Line.A1.Manual[#ConveyorID] := #ReadConveyorStatus.Manual;
	            DB_Global.Status.Line.A1.Stop[#ConveyorID] := #ReadConveyorStatus.Stop;
	            DB_Global.Status.Line.A1.Blockage[#ConveyorID] := #ReadConveyorStatus.Blockage;
	        END_IF;
	        // Line B1
	        IF #Active.Line.B1 THEN
	            DB_Global.Status.Line.B1.On[#ConveyorID] := #ReadConveyorStatus.ON;
	            DB_Global.Status.Line.B1.ReadyToRun[#ConveyorID] := #ReadConveyorStatus.ReadytoRun;
	            DB_Global.Status.Line.B1.Occupied[#ConveyorID] := #ReadConveyorStatus.Occupied;
	            DB_Global.Status.Line.B1.Running[#ConveyorID] := #ReadConveyorStatus.Running;
	            DB_Global.Status.Line.B1.Fault[#ConveyorID] := #ReadConveyorStatus.Fault;
	            DB_Global.Status.Line.B1.Estop[#ConveyorID] := #ReadConveyorStatus.Estop;
	            DB_Global.Status.Line.B1.Manual[#ConveyorID] := #ReadConveyorStatus.Manual;
	            DB_Global.Status.Line.B1.Stop[#ConveyorID] := #ReadConveyorStatus.Stop;
	            DB_Global.Status.Line.B1.Blockage[#ConveyorID] := #ReadConveyorStatus.Blockage;
	        END_IF;
	        // Line C1
	        IF #Active.Line.C1 THEN
	            DB_Global.Status.Line.C1.On[#ConveyorID] := #ReadConveyorStatus.ON;
	            DB_Global.Status.Line.C1.ReadyToRun[#ConveyorID] := #ReadConveyorStatus.ReadytoRun;
	            DB_Global.Status.Line.C1.Occupied[#ConveyorID] := #ReadConveyorStatus.Occupied;
	            DB_Global.Status.Line.C1.Running[#ConveyorID] := #ReadConveyorStatus.Running;
	            DB_Global.Status.Line.C1.Fault[#ConveyorID] := #ReadConveyorStatus.Fault;
	            DB_Global.Status.Line.C1.Estop[#ConveyorID] := #ReadConveyorStatus.Estop;
	            DB_Global.Status.Line.C1.Manual[#ConveyorID] := #ReadConveyorStatus.Manual;
	            DB_Global.Status.Line.C1.Stop[#ConveyorID] := #ReadConveyorStatus.Stop;
	            DB_Global.Status.Line.C1.Blockage[#ConveyorID] := #ReadConveyorStatus.Blockage;
	        END_IF;
	        // Line D1
	        IF #Active.Line.D1 THEN
	            DB_Global.Status.Line.D1.On[#ConveyorID] := #ReadConveyorStatus.ON;
	            DB_Global.Status.Line.D1.ReadyToRun[#ConveyorID] := #ReadConveyorStatus.ReadytoRun;
	            DB_Global.Status.Line.D1.Occupied[#ConveyorID] := #ReadConveyorStatus.Occupied;
	            DB_Global.Status.Line.D1.Running[#ConveyorID] := #ReadConveyorStatus.Running;
	            DB_Global.Status.Line.D1.Fault[#ConveyorID] := #ReadConveyorStatus.Fault;
	            DB_Global.Status.Line.D1.Estop[#ConveyorID] := #ReadConveyorStatus.Estop;
	            DB_Global.Status.Line.D1.Manual[#ConveyorID] := #ReadConveyorStatus.Manual;
	            DB_Global.Status.Line.D1.Stop[#ConveyorID] := #ReadConveyorStatus.Stop;
	            DB_Global.Status.Line.D1.Blockage[#ConveyorID] := #ReadConveyorStatus.Blockage;
	        END_IF;
	        
	    END_REGION
	    
	END_REGION
	
	REGION Run/Stop Conveyor 
	    
	    // FB_ConveyorRunStop
	    // Called as MIDB
	    
	    #"RUN/STOP_CONVEYOR"(StatusReady  := #ReadConveyorStatus.ReadytoRun,
	                         StatusOccu   := #ReadConveyorStatus.Occupied,
	                         DSOcc        := #Downstream,
	                         USOcc        := #Upstream,
	                         EnergySave   := #EnergySave,
	                         ILStop       := #Interlock,
	                         PecBlockage  := #ConveyorFault.Sensor_Blockage,
	                         MotorForward => #StartMotorForward,
	                         MotorReverse => #StartMotorReverse);
	    
	END_REGION
	
	REGION Energy Save
	    
	    // FB_EnergySave
	    // Called as MIDB
	    
	    #ENERGY_SAVE(StatusReady      := #ReadConveyorStatus.ReadytoRun,
	                 StatusOccupied   := #ReadConveyorStatus.Occupied,
	                 StartUpIN        := #SetStartUp,
	                 USOcc            := #Upstream,
	                 EnergySaveTimePT := #ReadConveyorParameters.EnergySaveTime,
	                 EnergySaveOut    => #EnergySave);
	    
	END_REGION
	
	REGION Write logic and parameters
	    
	    // Motor Forward: motors which has only one control bit
	    // Line A1 
	    IF #Active.Line.A1 THEN
	        #RunForward :=
	        (#StartMotorForward AND NOT #StartMotorReverse) // Automatic mode
	        OR (#ReadConveyorStatus.Manual AND DB_Manual.Line.A1.Conveyor[#ConveyorID].Run.Forward); //Manual mode
	    END_IF;
	    // Line B1 
	    IF #Active.Line.B1 THEN
	        #RunForward :=
	        (#StartMotorForward AND NOT #StartMotorReverse) // Automatic mode
	        OR (#ReadConveyorStatus.Manual AND DB_Manual.Line.B1.Conveyor[#ConveyorID].Run.Forward); //Manual mode
	    END_IF;
	    // Line C1 
	    IF #Active.Line.C1 THEN
	        #RunForward :=
	        (#StartMotorForward AND NOT #StartMotorReverse) // Automatic mode
	        OR (#ReadConveyorStatus.Manual AND DB_Manual.Line.C1.Conveyor[#ConveyorID].Run.Forward); //Manual mode
	    END_IF;
	    // Line D1 
	    IF #Active.Line.D1 THEN
	        #RunForward :=
	        (#StartMotorForward AND NOT #StartMotorReverse) // Automatic mode
	        OR (#ReadConveyorStatus.Manual AND DB_Manual.Line.D1.Conveyor[#ConveyorID].Run.Forward); //Manual mode
	    END_IF;
	    
	    REGION Bihl Wiedemann 
	        
	        // process data for BW-ASi
	        
	        IF #MotorType."24v-ASi" THEN
	            
	            REGION Direction
	                
	                // line A1
	                IF #Active.Line.A1 THEN
	                    #WriteAsiDir := DB_AsiSetpoint.Line.A1.DirChange.Conveyor[#ConveyorID];
	                END_IF;
	                // line B1
	                IF #Active.Line.B1 THEN
	                    #WriteAsiDir := DB_AsiSetpoint.Line.B1.DirChange.Conveyor[#ConveyorID];
	                END_IF;
	                // line C1
	                IF #Active.Line.C1 THEN
	                    #WriteAsiDir := DB_AsiSetpoint.Line.C1.DirChange.Conveyor[#ConveyorID];
	                END_IF;
	                // line D1
	                IF #Active.Line.D1 THEN
	                    #WriteAsiDir := DB_AsiSetpoint.Line.D1.DirChange.Conveyor[#ConveyorID];
	                END_IF;
	                
	            END_REGION
	            
	            REGION Speed
	                
	                // line A1
	                IF #Active.Line.A1 THEN
	                    #WriteAsiSpeed := DB_AsiSetpoint.Line.A1.Speed.Conveyor[#ConveyorID];
	                END_IF;
	                // line B1
	                IF #Active.Line.B1 THEN
	                    #WriteAsiSpeed := DB_AsiSetpoint.Line.B1.Speed.Conveyor[#ConveyorID];
	                END_IF;
	                // line C1
	                IF #Active.Line.C1 THEN
	                    #WriteAsiSpeed := DB_AsiSetpoint.Line.C1.Speed.Conveyor[#ConveyorID];
	                END_IF;
	                // line D1
	                IF #Active.Line.D1 THEN
	                    #WriteAsiSpeed := DB_AsiSetpoint.Line.D1.Speed.Conveyor[#ConveyorID];
	                END_IF;
	                
	            END_REGION
	            
	        END_IF;
	        
	    END_REGION
	    
	    REGION NORD (Line shaft)
	        
	        // process data and logic for NORD VFD
	        
	        IF #MotorType.nord THEN
	            
	            // Line A1
	            IF #Active.Line.A1 THEN
	                
	                IF NOT #ReadConveyorStatus.Fault THEN
	                    IF // Nord Motor Run - Automatic mode
	                        ((#ReadConveyorStatus.ReadytoRun AND
	                        #StartMotorForward) OR
	                        // Nord Motor Run - manual mode
	                        (#ReadConveyorStatus.Manual AND
	                        DB_Manual.Line.A1.Conveyor[#ConveyorID].Run.Forward))
	                    THEN
	                        #NordControlEnable := #NordSetpointRun;
	                    ELSE
	                        #NordControlEnable := #NordSetpointReady;
	                    END_IF;
	                END_IF;
	                
	                // Nord Motor Fault ack
	                IF #ReadConveyorStatus.Fault AND #SSR.ResetSystem THEN
	                    #NordControlEnable := #NordFaultAck;
	                END_IF;
	                
	                // Nord setpoint
	                #NordSetpoint := DINT_TO_WORD(DB_NordSetPoint.Line.A1.Conveyor[#ConveyorID]);
	                
	            END_IF;
	            
	            // Line B1
	            IF #Active.Line.B1 THEN
	                
	                IF NOT #ReadConveyorStatus.Fault THEN
	                    IF // Nord Motor Run - Automatic mode
	                        ((#ReadConveyorStatus.ReadytoRun AND
	                        #StartMotorForward) OR
	                        // Nord Motor Run - manual mode
	                        (#ReadConveyorStatus.Manual AND
	                        DB_Manual.Line.B1.Conveyor[#ConveyorID].Run.Forward))
	                    THEN
	                        #NordControlEnable := #NordSetpointRun;
	                    ELSE
	                        #NordControlEnable := #NordSetpointReady;
	                    END_IF;
	                END_IF;
	                
	                // Nord Motor Fault ack
	                IF #ReadConveyorStatus.Fault AND #SSR.ResetSystem THEN
	                    #NordControlEnable := #NordFaultAck;
	                END_IF;
	                
	                // Nord setpoint
	                #NordSetpoint := DINT_TO_WORD(DB_NordSetPoint.Line.B1.Conveyor[#ConveyorID]);
	                
	            END_IF;
	            
	            // Line C1
	            IF #Active.Line.C1 THEN
	                
	                IF NOT #ReadConveyorStatus.Fault THEN
	                    IF // Nord Motor Run - Automatic mode
	                        ((#ReadConveyorStatus.ReadytoRun AND
	                        #StartMotorForward) OR
	                        // Nord Motor Run - manual mode
	                        (#ReadConveyorStatus.Manual AND
	                        DB_Manual.Line.C1.Conveyor[#ConveyorID].Run.Forward))
	                    THEN
	                        #NordControlEnable := #NordSetpointRun;
	                    ELSE
	                        #NordControlEnable := #NordSetpointReady;
	                    END_IF;
	                END_IF;
	                
	                // Nord Motor Fault ack
	                IF #ReadConveyorStatus.Fault AND #SSR.ResetSystem THEN
	                    #NordControlEnable := #NordFaultAck;
	                END_IF;
	                
	                // Nord setpoint
	                #NordSetpoint := DINT_TO_WORD(DB_NordSetPoint.Line.C1.Conveyor[#ConveyorID]);
	                
	            END_IF;
	            
	            // Line D1
	            IF #Active.Line.D1 THEN
	                
	                IF NOT #ReadConveyorStatus.Fault THEN
	                    IF // Nord Motor Run - Automatic mode
	                        ((#ReadConveyorStatus.ReadytoRun AND
	                        #StartMotorForward) OR
	                        // Nord Motor Run - manual mode
	                        (#ReadConveyorStatus.Manual AND
	                        DB_Manual.Line.D1.Conveyor[#ConveyorID].Run.Forward))
	                    THEN
	                        #NordControlEnable := #NordSetpointRun;
	                    ELSE
	                        #NordControlEnable := #NordSetpointReady;
	                    END_IF;
	                END_IF;
	                
	                // Nord Motor Fault ack
	                IF #ReadConveyorStatus.Fault AND #SSR.ResetSystem THEN
	                    #NordControlEnable := #NordFaultAck;
	                END_IF;
	                
	                // Nord setpoint
	                #NordSetpoint := DINT_TO_WORD(DB_NordSetPoint.Line.D1.Conveyor[#ConveyorID]);
	                
	            END_IF;
	            
	        END_IF;
	        
	    END_REGION
	    
	END_REGION
	
END_FUNCTION_BLOCK
END_NAMESPACE

NAMESPACE Global
FUNCTION_BLOCK FB_MABS
{ S7_Optimized_Access := 'TRUE' ; Published := 'TRUE' }
VERSION : 0.1
   VAR_INPUT 
      MABS_ID : Int;
      CrossSensor : Bool;
      Fault : Bool;
      UpstreamRunning : Bool;
      Downstream_Straight : Bool;
      "Downstream_Right/Left" : Bool;
      SortDir : ItemDir;
      ManIn : MABS_ManIn;
      Setpoints : MABS_Setpoint;
   END_VAR

   VAR_IN_OUT 
      MABS_IBP_in : _."IB_P01/02/03_in_64bytes_struct";
      MABS_IBP_out : _."IB_P01/02/03_out_64bytes_struct";
   END_VAR

   VAR 
      ReadInputSignal : Struct
         CrossSensor : Bool;
         EmergencyStop : Bool;
         Fault : Bool;
      END_STRUCT;
      Active : Struct
         Line : Struct
            A1 : Bool;
            B1 : Bool;
            C1 : Bool;
            D1 : Bool;
         END_STRUCT;
      END_STRUCT;
      CROSS_SENSOR_FILTER : FB_Sensor;
      MABS_SENSOR_BLOCKAGE {InstructionName := 'IEC_TIMER'; LibVersion := '1.0'} : IEC_TIMER;
      MABS_STATUS_ON : FB_StatusON;
      MABS_STATUS_READY : FB_StatusReady;
      MABS_STATUS_FAULT : FB_StatusFault;
      AUTO_RESET : FB_AutoReset;
      MABS_CONTROL : FB_MABS_PNIO;
      SSR : SystemSSR;
      ReadMabsStatus : ConveyorStatus;
      ReadMabsParameter : ConveyorParameters := ((), [2(T#10ms)], (), (), ());
      MABSFault : Fault;
      SimuMode : Struct
         Sensor : Bool;
         Fault : Bool;
      END_STRUCT;
      StartUpTimer {InstructionName := 'TOF_TIME'; LibVersion := '1.0'; S7_SetPoint := 'False'} : TOF_TIME;
      FT_StartUp {InstructionName := 'F_TRIG'; LibVersion := '1.0'} : F_TRIG;
      SetStartUp { S7_SetPoint := 'True'} : Bool;
      VisuColor : Word;
      PhaseError : Bool;
      StartupMABS { S7_SetPoint := 'True'} : Bool;
      FilteredSensor { S7_SetPoint := 'True'} : Bool;
      AutoReset { S7_SetPoint := 'True'} : Bool;
      StopSystemFireActive : Bool;
      Sort { S7_SetPoint := 'False'} : ItemDir;
      Home : Bool;
      HomeCheckTimer {InstructionName := 'TON_TIME'; LibVersion := '1.0'} : TON_TIME;
      CurrentPosition : Struct
         left : Bool;
         right : Bool;
         straight : Bool;
      END_STRUCT;
      "Cmd+Setpoint" { ExternalAccessible := 'False'; ExternalVisible := 'False'; ExternalWritable := 'False'; S7_SetPoint := 'False'} : MABS;
   END_VAR


BEGIN
	// ==========================================================================================================================================
	// Company        : LogTech, s.r.o.
	// Created by     : Anton Vinoth Soundraraj
	// Block          : FB_MABS
	// Project        : Lékarna DC Chrudim
	// Project number : 23-157
	// ==========================================================================================================================================
	
	REGION Active Line
	    
	    // Line A1
	    IF (#MABS_ID >= _.gMinA1 AND
	        #MABS_ID <= _.gMaxA1)
	    THEN
	        #Active.Line.A1 := TRUE;
	    END_IF;
	    
	    // Line B1
	    IF (#MABS_ID >= _.gMinB1 AND
	        #MABS_ID <= _.gMaxB1)
	    THEN
	        #Active.Line.B1 := TRUE;
	    END_IF;
	    
	    // Line C1
	    IF (#MABS_ID >= _.gMinC1 AND
	        #MABS_ID <= _.gMaxC1)
	    THEN
	        #Active.Line.C1 := TRUE;
	    END_IF;
	    
	    // Line D1
	    IF (#MABS_ID >= _.gMinD1 AND
	        #MABS_ID <= _.gMaxD1)
	    THEN
	        #Active.Line.A1 := TRUE;
	    END_IF;
	    
	END_REGION
	
	REGION SystemSSR
	    
	    // Line A1
	    IF #Active.Line.A1 THEN
	        #SSR.StartSystem := DB_SystemSSR.Line.A1.StartSystem;
	        #SSR.StopSystem := DB_SystemSSR.Line.A1.StopSystem;
	        #SSR.ResetSystem := DB_SystemSSR.Line.A1.ResetSystem;
	    END_IF;
	    
	    // Line B1
	    IF #Active.Line.B1 THEN
	        #SSR.StartSystem := DB_SystemSSR.Line.B1.StartSystem;
	        #SSR.StopSystem := DB_SystemSSR.Line.B1.StopSystem;
	        #SSR.ResetSystem := DB_SystemSSR.Line.B1.ResetSystem;
	    END_IF;
	    
	    // Line C1
	    IF #Active.Line.C1 THEN
	        #SSR.StartSystem := DB_SystemSSR.Line.C1.StartSystem;
	        #SSR.StopSystem := DB_SystemSSR.Line.C1.StopSystem;
	        #SSR.ResetSystem := DB_SystemSSR.Line.C1.ResetSystem;
	    END_IF;
	    
	    // Line D1
	    IF #Active.Line.D1 THEN
	        #SSR.StartSystem := DB_SystemSSR.Line.D1.StartSystem;
	        #SSR.StopSystem := DB_SystemSSR.Line.D1.StopSystem;
	        #SSR.ResetSystem := DB_SystemSSR.Line.D1.ResetSystem;
	    END_IF;
	    
	END_REGION
	
	REGION Read Input
	    
	    // read all inputs to the block
	    // Conveyor input read signals
	    #ReadInputSignal.CrossSensor := NOT #CrossSensor OR
	    #SimuMode.Sensor; // simu call
	    #ReadInputSignal.Fault := #Fault OR
	    #SimuMode.Fault; // simu call;
	    #ReadInputSignal.EmergencyStop := // all estop zones are connected together
	    _.DB_SafetyStandard.ToStandard.EstopActive;
	    
	END_REGION
	
	REGION READ AND INIT
	    
	    REGION parameters
	        
	        // Line A1
	        IF #Active.Line.A1 THEN
	            #ReadMabsParameter := DB_ConveyorParameters.Line.A1.Conveyor[#MABS_ID];
	        END_IF;
	        // Line B1
	        IF #Active.Line.B1 THEN
	            #ReadMabsParameter := DB_ConveyorParameters.Line.B1.Conveyor[#MABS_ID];
	        END_IF;
	        // Line C1
	        IF #Active.Line.C1 THEN
	            #ReadMabsParameter := DB_ConveyorParameters.Line.C1.Conveyor[#MABS_ID];
	        END_IF;
	        // Line C1
	        IF #Active.Line.D1 THEN
	            #ReadMabsParameter := DB_ConveyorParameters.Line.D1.Conveyor[#MABS_ID];
	        END_IF;
	        
	    END_REGION
	    
	    REGION FIRE
	        
	        // Fire signal from fire system stops the whole system
	        // System can be reset from Fire status only if the fire signal is deactivated
	        
	        // FIRE ALARM ACTIVE --> STOP SYSTEM
	        IF DB_SystemSimu.Fire THEN
	            #StopSystemFireActive := TRUE;
	        END_IF;
	        // RESET --> FIRE ALARM
	        IF #SSR.ResetSystem AND NOT DB_SystemSimu.Fire THEN
	            #StopSystemFireActive := FALSE;
	        END_IF;
	        
	    END_REGION
	    
	END_REGION
	
	REGION Conveyor startup
	    
	    // Conveyor StartUp: Conveyor startup signal after 5 second delay
	    
	    #StartUpTimer.TOF(IN := #SSR.StartSystem,
	                      PT := #ReadMabsParameter.StartUpTime);
	    
	    #FT_StartUp(CLK := #StartUpTimer.Q);
	    
	    // set startup after 5 seconds
	    #SetStartUp := #FT_StartUp.Q;
	    
	END_REGION
	
	REGION Conveyor Status
	    
	    REGION Status ON
	        
	        // ----------------------------------------->>>>>>> STATUS ON <<<<<<<-----------------------------------------
	        // FB_ConveyorStatusON
	        // called as IDMB
	        
	        #MABS_STATUS_ON(SystemStartActive := #SSR.StartSystem,
	                        StatusStop := #ReadMabsStatus.Stop,
	                        StatusEStop := #ReadMabsStatus.Estop,
	                        StatusManual := #ReadMabsStatus.Manual,
	                        StatusFault := #ReadMabsStatus.Fault,
	                        FireAlarmActive := #StopSystemFireActive,
	                        StatusON => #ReadMabsStatus.ON);
	        
	    END_REGION
	    
	    REGION Status Ready
	        
	        // ----------------------------------------->>>>>>> STATUS READY <<<<<<<-----------------------------------------
	        // FB_ConveyorStatusReady
	        // called as MIDB
	        
	        #MABS_STATUS_READY(StatusON := #ReadMabsStatus.ON,
	                           StatusESTOP := #ReadMabsStatus.Estop,
	                           StatusFAULT := #ReadMabsStatus.Fault,
	                           StatusMAN := #ReadMabsStatus.Manual,
	                           SignalFIRE := #StopSystemFireActive,
	                           SystemAlertTime := #ReadMabsParameter.StartUpTime,
	                           StatusReady => #ReadMabsStatus.ReadytoRun);
	        
	    END_REGION
	    
	    REGION Status Occupied
	        
	        // ----------------------------------------->>>>>>> STATUS OCCUPIED <<<<<<<-----------------------------------------
	        
	        #ReadMabsStatus.Occupied :=
	        #CROSS_SENSOR_FILTER.FilteredSensor;
	        
	    END_REGION
	    
	    REGION Status Running
	        
	        // ----------------------------------------->>>>>>> STATUS RUNNING <<<<<<<-----------------------------------------
	        
	        #ReadMabsStatus.Running :=
	        #ReadMabsStatus.ReadytoRun AND
	        #"Cmd+Setpoint".Run_balls;
	        
	    END_REGION
	    
	    REGION Status Fault
	        
	        // ----------------------------------------->>>>>>> STATUS FAULT <<<<<<<-----------------------------------------
	        
	        // Reading error signal from the motor drive
	        #MABSFault.Motor_Error := #ReadInputSignal.Fault;
	        
	        // FC_ConveyorStatusFault
	        #MABS_STATUS_FAULT(FaultActive := #MABSFault.Motor_Error,
	                           ResetFault := #SSR.ResetSystem,
	                           StatusRunning := #ReadMabsStatus.Running,
	                           FaultStatus => #ReadMabsStatus.Fault);
	        
	    END_REGION
	    
	    REGION Status ESTOP
	        
	        // ----------------------------------------->>>>>>> STATUS ESTOP <<<<<<<-----------------------------------------
	        
	        #AUTO_RESET(AckIN := #SSR.ResetSystem,
	                    Ack => #AutoReset);
	        
	        // EMERGENCY STOP ACTIVE --> STOP SYSTEM
	        IF #ReadInputSignal.EmergencyStop THEN
	            #ReadMabsStatus.Estop := TRUE;
	        END_IF;
	        // RESET --> EMERGENCY STOP
	        IF #AutoReset AND NOT #ReadInputSignal.EmergencyStop THEN
	            #ReadMabsStatus.Estop := FALSE;
	        END_IF;
	        
	    END_REGION
	    
	    REGION Status Stop
	        
	        // ----------------------------------------->>>>>>> STATUS STOP <<<<<<<-----------------------------------------
	        
	        IF #SSR.StopSystem THEN
	            #ReadMabsStatus.Stop := TRUE;
	        END_IF;
	        IF #SSR.StartSystem OR #SSR.ResetSystem THEN
	            #ReadMabsStatus.Stop := FALSE;
	        END_IF;
	        
	    END_REGION
	    
	    REGION Sensor Blockage
	        
	        // ----------------------------------------->>>>>>> STATUS BLOCKAGE <<<<<<<-------------------------------------
	        
	        // FB_SensorBlockage
	        // called as MIDB
	        
	        #MABS_SENSOR_BLOCKAGE.TON(IN := #ReadMabsStatus.ReadytoRun AND
	                                  #CROSS_SENSOR_FILTER.FilteredSensor,
	                                  PT := #ReadMabsParameter.SensorBlockageTime,
	                                  Q => #ReadMabsStatus.Blockage);
	        
	        // ==========================
	        // Sensor Blockage: HMI Alarm
	        // ==========================
	        // Sensor blockage alarm message is written to the first bit of the alarm word
	        // corresponding to the active line
	        
	        REGION alarm 
	            
	            // ==========================
	            // Sensor Blockage: HMI Alarm
	            // ==========================
	            // Sensor blockage alarm message is written to the alarm word
	            // corresponding to the active line
	            // Line A1
	            IF #Active.Line.A1 THEN
	                DB_Alarm."word".Line.A1.Conveyor[#MABS_ID].%X0 := #ReadMabsStatus.Blockage;
	            END_IF;
	            // Line B1
	            IF #Active.Line.B1 THEN
	               DB_Alarm."word".Line.B1.Conveyor[#MABS_ID].%X0 := #ReadMabsStatus.Blockage;
	            END_IF;
	            // Line C1
	            IF #Active.Line.C1 THEN
	               DB_Alarm."word".Line.C1.Conveyor[#MABS_ID].%X0 := #ReadMabsStatus.Blockage;
	            END_IF;
	            // Line D1
	            IF #Active.Line.D1 THEN
	                DB_Alarm."word".Line.D1.Conveyor[#MABS_ID].%X0 := #ReadMabsStatus.Blockage;
	            END_IF;
	            
	        END_REGION
	        
	    END_REGION
	    
	    REGION Visu Color
	        
	        // each and every status of the conveyor will be mentioned by different colors in HMI panel
	        
	        #VisuColor.%X8 := #ReadMabsStatus.Blockage;
	        #VisuColor.%X0 := #ReadMabsStatus.ON;
	        #VisuColor.%X1 := #ReadMabsStatus.ReadytoRun;
	        #VisuColor.%X2 := #ReadMabsStatus.Occupied;
	        #VisuColor.%X3 := #ReadMabsStatus.Running;
	        #VisuColor.%X4 := #ReadMabsStatus.Fault;
	        #VisuColor.%X5 := #ReadMabsStatus.Estop;
	        #VisuColor.%X6 := #ReadMabsStatus.Manual;
	        #VisuColor.%X7 := #ReadMabsStatus.Stop;
	        
	        // convert word to Interger value: 
	        // color will be depends on the status priority (integer value) 
	        // reference: Conveyor image in HMI screen -> property -> Apperance   
	        
	        // Line A1
	        IF #Active.Line.A1 THEN
	            DB_VisuColor.Line.A1.Conveyor[#MABS_ID] :=
	            WORD_TO_INT(#VisuColor);
	        END_IF;
	        // Line B1
	        IF #Active.Line.B1 THEN
	            DB_VisuColor.Line.B1.Conveyor[#MABS_ID] :=
	            WORD_TO_INT(#VisuColor);
	        END_IF;
	        // Line C1
	        IF #Active.Line.C1 THEN
	            DB_VisuColor.Line.C1.Conveyor[#MABS_ID] :=
	            WORD_TO_INT(#VisuColor);
	        END_IF;
	        // Line D1
	        IF #Active.Line.D1 THEN
	            DB_VisuColor.Line.D1.Conveyor[#MABS_ID] :=
	            WORD_TO_INT(#VisuColor);
	        END_IF;
	        
	    END_REGION
	    
	    REGION Global Status
	        
	        // write -> global status
	        // Line A1
	        IF #Active.Line.A1 THEN
	            DB_Global.Status.Line.A1.On[#MABS_ID] := #ReadMabsStatus.ON;
	            DB_Global.Status.Line.A1.ReadyToRun[#MABS_ID] := #ReadMabsStatus.ReadytoRun;
	            DB_Global.Status.Line.A1.Occupied[#MABS_ID] := #ReadMabsStatus.Occupied;
	            DB_Global.Status.Line.A1.Running[#MABS_ID] := #ReadMabsStatus.Running;
	            DB_Global.Status.Line.A1.Fault[#MABS_ID] := #ReadMabsStatus.Fault;
	            DB_Global.Status.Line.A1.Estop[#MABS_ID] := #ReadMabsStatus.Estop;
	            DB_Global.Status.Line.A1.Manual[#MABS_ID] := #ReadMabsStatus.Manual;
	            DB_Global.Status.Line.A1.Stop[#MABS_ID] := #ReadMabsStatus.Stop;
	            DB_Global.Status.Line.A1.Blockage[#MABS_ID] := #ReadMabsStatus.Blockage;
	        END_IF;
	        // Line B1
	        IF #Active.Line.B1 THEN
	            DB_Global.Status.Line.B1.On[#MABS_ID] := #ReadMabsStatus.ON;
	            DB_Global.Status.Line.B1.ReadyToRun[#MABS_ID] := #ReadMabsStatus.ReadytoRun;
	            DB_Global.Status.Line.B1.Occupied[#MABS_ID] := #ReadMabsStatus.Occupied;
	            DB_Global.Status.Line.B1.Running[#MABS_ID] := #ReadMabsStatus.Running;
	            DB_Global.Status.Line.B1.Fault[#MABS_ID] := #ReadMabsStatus.Fault;
	            DB_Global.Status.Line.B1.Estop[#MABS_ID] := #ReadMabsStatus.Estop;
	            DB_Global.Status.Line.B1.Manual[#MABS_ID] := #ReadMabsStatus.Manual;
	            DB_Global.Status.Line.B1.Stop[#MABS_ID] := #ReadMabsStatus.Stop;
	            DB_Global.Status.Line.B1.Blockage[#MABS_ID] := #ReadMabsStatus.Blockage;
	        END_IF;
	        // Line C1
	        IF #Active.Line.C1 THEN
	            DB_Global.Status.Line.C1.On[#MABS_ID] := #ReadMabsStatus.ON;
	            DB_Global.Status.Line.C1.ReadyToRun[#MABS_ID] := #ReadMabsStatus.ReadytoRun;
	            DB_Global.Status.Line.C1.Occupied[#MABS_ID] := #ReadMabsStatus.Occupied;
	            DB_Global.Status.Line.C1.Running[#MABS_ID] := #ReadMabsStatus.Running;
	            DB_Global.Status.Line.C1.Fault[#MABS_ID] := #ReadMabsStatus.Fault;
	            DB_Global.Status.Line.C1.Estop[#MABS_ID] := #ReadMabsStatus.Estop;
	            DB_Global.Status.Line.C1.Manual[#MABS_ID] := #ReadMabsStatus.Manual;
	            DB_Global.Status.Line.C1.Stop[#MABS_ID] := #ReadMabsStatus.Stop;
	            DB_Global.Status.Line.C1.Blockage[#MABS_ID] := #ReadMabsStatus.Blockage;
	        END_IF;
	        // Line D1
	        IF #Active.Line.D1 THEN
	            DB_Global.Status.Line.D1.On[#MABS_ID] := #ReadMabsStatus.ON;
	            DB_Global.Status.Line.D1.ReadyToRun[#MABS_ID] := #ReadMabsStatus.ReadytoRun;
	            DB_Global.Status.Line.D1.Occupied[#MABS_ID] := #ReadMabsStatus.Occupied;
	            DB_Global.Status.Line.D1.Running[#MABS_ID] := #ReadMabsStatus.Running;
	            DB_Global.Status.Line.D1.Fault[#MABS_ID] := #ReadMabsStatus.Fault;
	            DB_Global.Status.Line.D1.Estop[#MABS_ID] := #ReadMabsStatus.Estop;
	            DB_Global.Status.Line.D1.Manual[#MABS_ID] := #ReadMabsStatus.Manual;
	            DB_Global.Status.Line.D1.Stop[#MABS_ID] := #ReadMabsStatus.Stop;
	            DB_Global.Status.Line.D1.Blockage[#MABS_ID] := #ReadMabsStatus.Blockage;
	        END_IF;
	        
	    END_REGION
	    
	END_REGION
	
	REGION Sorter sensor filter
	    
	    // cross sensor filter
	    #CROSS_SENSOR_FILTER(Sensor := #CrossSensor,
	                         SensorFilterTime := #ReadMabsParameter.SensorFilterTime,
	                         FilteredSensor=>#FilteredSensor);
	END_REGION
	
	REGION MABS LOGIC
	    
	    REGION rcv direction 
	        
	        IF NOT #FilteredSensor THEN
	            #Sort := #SortDir;
	        END_IF;
	        
	    END_REGION
	    
	    REGION MABS lib block
	        
	        #MABS_CONTROL(IBP_in  := #MABS_IBP_in,
	                      IBP_out := #MABS_IBP_out,
	                      MABS    := #"Cmd+Setpoint");
	        
	    END_REGION
	    
	    REGION run MABS wheels
	        
	        #"Cmd+Setpoint".Run_balls := #UpstreamRunning;
	        
	    END_REGION
	    
	    REGION Current position
	        
	        #CurrentPosition.left := #"Cmd+Setpoint".Left_Pos_reach;
	        #CurrentPosition.right := #"Cmd+Setpoint".Right_Pos_reach;
	        #CurrentPosition.straight := #"Cmd+Setpoint".Straight_Pos_reach;
	        
	    END_REGION
	    
	    REGION HOMING
	        
	        // ==========================================================================================================================
	        // Initial operation (home searching)
	        // ==================================
	        
	        // Home missing (if MABS could not receive any position in 't' duration)
	        #HomeCheckTimer.TON(IN := NOT #CurrentPosition.left AND
	                            NOT #CurrentPosition.right AND
	                            NOT #CurrentPosition.straight,
	                            PT := T#2s);
	        #Home :=
	        NOT #HomeCheckTimer.Q;
	        
	        // init HOME
	        IF NOT #Home AND NOT #ReadMabsStatus.Stop THEN
	            #"Cmd+Setpoint".Init := TRUE;
	        END_IF;
	        // RESET -> Init Home
	        IF #Home THEN
	            #"Cmd+Setpoint".Init := TRUE;
	        END_IF;
	        
	    END_REGION
	    
	    REGION Parameters
	        
	        // change balls direction
	        #"Cmd+Setpoint".Dir_balls := #Setpoints.ChangeBallsDirection;
	        // balls speed
	        #"Cmd+Setpoint".Speed_balls := #Setpoints.Speed_balls;
	        // offset for straight
	        #"Cmd+Setpoint".Init_offset := #Setpoints.Init_offset;
	        
	    END_REGION
	    
	    REGION Sorting logic
	        
	        IF #ReadMabsStatus.ReadytoRun
	        THEN
	            
	            REGION Straight
	                
	                // ================================================== ^^^
	                
	                // sort straight - actual position: right
	                
	                IF #Sort.Straight AND
	                    NOT #CurrentPosition.straight AND
	                    #CurrentPosition.right AND
	                    NOT #CROSS_SENSOR_FILTER.FilteredSensor
	                THEN
	                    #"Cmd+Setpoint".Switch_right_to_st := TRUE;
	                ELSE
	                    #"Cmd+Setpoint".Switch_right_to_st := FALSE;
	                END_IF;
	                
	                // sort straight - actual position: left
	                
	                IF #Sort.Straight AND
	                    NOT #CurrentPosition.straight AND
	                    #CurrentPosition.left AND
	                    NOT #CROSS_SENSOR_FILTER.FilteredSensor
	                THEN
	                    #"Cmd+Setpoint".Switch_left_to_st := TRUE;
	                ELSE
	                    #"Cmd+Setpoint".Switch_left_to_st := FALSE;
	                END_IF;
	                
	            END_REGION
	            
	            REGION to Right
	                
	                // ================================================== >>>
	                
	                // sort right - actual position: straight/left
	                
	                IF #Sort.toRight AND
	                    NOT #CurrentPosition.right AND
	                    (#CurrentPosition.straight OR
	                    #CurrentPosition.left) AND
	                    NOT #CROSS_SENSOR_FILTER.FilteredSensor
	                THEN
	                    #"Cmd+Setpoint".Switch_right := TRUE;
	                ELSE
	                    #"Cmd+Setpoint".Switch_right := FALSE;
	                END_IF;
	                
	            END_REGION
	            
	            REGION to left
	                
	                // ================================================== <<<
	                
	                // sort left - actual position: straight/right
	                
	                IF #Sort.toLeft AND
	                    NOT #CurrentPosition.left AND
	                    (#CurrentPosition.straight OR
	                    #CurrentPosition.right) AND
	                    NOT #CROSS_SENSOR_FILTER.FilteredSensor
	                THEN
	                    #"Cmd+Setpoint".Switch_left := TRUE;
	                ELSE
	                    #"Cmd+Setpoint".Switch_left := FALSE;
	                END_IF;
	                
	            END_REGION
	            
	            // ============================================================================================================
	            
	        END_IF;
	        
	    END_REGION
	    
	   REGION reset error 
	        
	        // reset error
	       IF #ReadMabsStatus.Fault AND
	           #SSR.ResetSystem
	       THEN
	            #"Cmd+Setpoint".Reset_error := TRUE;
	        ELSE
	            #"Cmd+Setpoint".Reset_error := FALSE;
	        END_IF;
	        
	    END_REGION
	    
	    REGION stop function
	        
	        // stop if not ready
	        IF NOT #ReadMabsStatus.ReadytoRun AND NOT #ReadMabsStatus.Manual
	        THEN
	            #"Cmd+Setpoint".Switch_left := FALSE;
	            #"Cmd+Setpoint".Switch_right := FALSE;
	            #"Cmd+Setpoint".Switch_right_to_st := FALSE;
	            #"Cmd+Setpoint".Switch_left_to_st := FALSE;
	        END_IF;
	        
	    END_REGION
	    
	END_REGION
	
	
	
END_FUNCTION_BLOCK
END_NAMESPACE

NAMESPACE Global
FUNCTION_BLOCK FB_S300_tTransMode
{ S7_Optimized_Access := 'TRUE' ; Published := 'TRUE' }
VERSION : 0.1
   VAR_INPUT 
      TransferID : Int;
      TransferSensor : Bool;
      Fault : Bool;
      ReadyToRCV : Bool;
      Upstream : Bool;
      FrontSensor : Bool;
      EndSensor : Bool;
      "Left/RightSensor" : Bool;
      Downstream : Bool;
      FrontSensorFilterTime : Array[1..2] of Time;
      TransferDirection : ItemDir;
   END_VAR

   VAR_OUTPUT 
      StartSignal : Bool;
      Cmd1 : Bool;
      Cmd2 : Bool;
      ErrorReset : Bool;
   END_VAR

   VAR 
      ReadInputSignal : Struct
         EmergencyStop : Bool;
         FireActive : Bool;
         Fault : Bool;
         TransferSensor : Bool;
      END_STRUCT;
      Active : Struct
         Line : Struct
            A1 : Bool;
            B1 : Bool;
            C1 : Bool;
            D1 : Bool;
         END_STRUCT;
      END_STRUCT;
      TRANSFER_SENSOR : FB_Sensor;
      FRONT_SENSOR_FILTER : FB_Sensor;
      TRANSFER_SENSOR_BLOCKAGE {InstructionName := 'TON_TIME'; LibVersion := '1.0'} : TON_TIME;
      FRONT_SENSOR_BLOCKAGE {InstructionName := 'TON_TIME'; LibVersion := '1.0'} : TON_TIME;
      END_SENSOR_BLOCKAGE {InstructionName := 'TON_TIME'; LibVersion := '1.0'} : TON_TIME;
      "LEFT/RIGHT_SENSOR_BLOCKAGE" {InstructionName := 'TON_TIME'; LibVersion := '1.0'} : TON_TIME;
      TRANSFER_STATUS_ON : FB_StatusON;
      TRANSFER_STATUS_READY : FB_StatusReady;
      TRANSFER_STATUS_FAULT : FB_StatusFault;
      AUTO_RESET : FB_AutoReset;
      StartUpTimer {InstructionName := 'TOF_TIME'; LibVersion := '1.0'; S7_SetPoint := 'False'} : TOF_TIME;
      FT_StartUp {InstructionName := 'F_TRIG'; LibVersion := '1.0'} : F_TRIG;
      SetStartUp { S7_SetPoint := 'True'} : Bool;
      Init : Struct
         Line : Struct
            A1 : String := 'LineA1';
         END_STRUCT;
      END_STRUCT;
      SSR : SystemSSR;
      ReadTransferStatus : ConveyorStatus;
      ReadTransferParameters : ConveyorParameters := ((), [2(T#10ms)], (), (), ());
      ConveyorFault : Fault;
      StartupTransfer { S7_SetPoint := 'True'} : Bool;
      FilteredSensor { S7_SetPoint := 'True'} : Bool;
      StopSystemFireActive : Bool;
      ClearTransferArea : Bool;
      AutoReset : Bool;
      VisuColor : Word;
      Transfer : Struct
         RcvInfeed : Bool;
         StartSignal : Bool;
         Command_1 : Bool;
         Command_2 : Bool;
      END_STRUCT;
      NegEdgeUpstream {InstructionName := 'F_TRIG'; LibVersion := '1.0'; S7_SetPoint := 'False'} : F_TRIG;
      CrossSensorFilterTime { S7_SetPoint := 'True'} : Array[0..1] of Time;
      sTransferDirection { S7_SetPoint := 'False'} : ItemDir;
   END_VAR


BEGIN
	// ==========================================================================================================================================
	// Company        : LogTech, s.r.o.
	// Created by     : Anton Vinoth Soundraraj
	// Block          : FB_S300_tTransMode
	// Project        : Lékarna DC Chrudim
	// Project number : 23-157
	// ==========================================================================================================================================
	
	REGION Active Line
	    
	    // Line A1
	    IF (#TransferID >= _.gMinA1 AND
	        #TransferID <= _.gMaxA1)
	    THEN
	        #Active.Line.A1 := TRUE;
	    END_IF;
	    
	    // Line B1
	    IF (#TransferID >= _.gMinB1 AND
	        #TransferID <= _.gMaxB1)
	    THEN
	        #Active.Line.B1 := TRUE;
	    END_IF;
	    
	    // Line C1
	    IF (#TransferID >= _.gMinC1 AND
	        #TransferID <= _.gMaxC1)
	    THEN
	        #Active.Line.C1 := TRUE;
	    END_IF;
	    
	    // Line D1
	    IF (#TransferID >= _.gMinD1 AND
	        #TransferID <= _.gMaxD1)
	    THEN
	        #Active.Line.A1 := TRUE;
	    END_IF;
	    
	END_REGION
	
	REGION SystemSSR
	    
	    // Line A1
	    IF #Active.Line.A1 THEN
	        #SSR.StartSystem := DB_SystemSSR.Line.A1.StartSystem;
	        #SSR.StopSystem := DB_SystemSSR.Line.A1.StopSystem;
	        #SSR.ResetSystem := DB_SystemSSR.Line.A1.ResetSystem;
	    END_IF;
	    
	    // Line B1
	    IF #Active.Line.B1 THEN
	        #SSR.StartSystem := DB_SystemSSR.Line.B1.StartSystem;
	        #SSR.StopSystem := DB_SystemSSR.Line.B1.StopSystem;
	        #SSR.ResetSystem := DB_SystemSSR.Line.B1.ResetSystem;
	    END_IF;
	    
	    // Line C1
	    IF #Active.Line.C1 THEN
	        #SSR.StartSystem := DB_SystemSSR.Line.C1.StartSystem;
	        #SSR.StopSystem := DB_SystemSSR.Line.C1.StopSystem;
	        #SSR.ResetSystem := DB_SystemSSR.Line.C1.ResetSystem;
	    END_IF;
	    
	    // Line D1
	    IF #Active.Line.D1 THEN
	        #SSR.StartSystem := DB_SystemSSR.Line.D1.StartSystem;
	        #SSR.StopSystem := DB_SystemSSR.Line.D1.StopSystem;
	        #SSR.ResetSystem := DB_SystemSSR.Line.D1.ResetSystem;
	    END_IF;
	    
	END_REGION
	
	REGION Read Input
	    
	    // read all inputs to the block
	    // Conveyor input read signals
	    #ReadInputSignal.TransferSensor := #TransferSensor;
	    #ReadInputSignal.Fault := #Fault;
	    // Read static tag connections
	    #ReadInputSignal.EmergencyStop := // all estop zones are connected together
	    _.DB_SafetyStandard.ToStandard.EstopActive;
	    // Common system input Read
	    #ReadInputSignal.FireActive :=
	    DB_SystemSimu.Fire; // simu call
	    
	END_REGION
	
	REGION Conveyor startup
	    
	    // Conveyor StartUp: Conveyor startup signal after preset time
	    #StartUpTimer.TOF(IN := #SSR.StartSystem,
	                      PT := #ReadTransferParameters.StartUpTime);
	    
	    #FT_StartUp(CLK := #StartUpTimer.Q);
	    
	    // set startup after the preset
	    #SetStartUp := #FT_StartUp.Q;
	    
	END_REGION
	
	REGION READ AND INIT
	    
	    REGION Init conveyor parameters
	        
	        // Conveyor Parameter
	        // Line A1
	        IF #Active.Line.A1 THEN
	            #ReadTransferParameters := DB_ConveyorParameters.Line.A1.Conveyor[#TransferID];
	        END_IF;
	        // Line B1
	        IF #Active.Line.B1 THEN
	            #ReadTransferParameters := DB_ConveyorParameters.Line.B1.Conveyor[#TransferID];
	        END_IF;
	        // Line C1
	        IF #Active.Line.C1 THEN
	            #ReadTransferParameters := DB_ConveyorParameters.Line.C1.Conveyor[#TransferID];
	        END_IF;
	        // Line D1
	        IF #Active.Line.D1 THEN
	            #ReadTransferParameters := DB_ConveyorParameters.Line.D1.Conveyor[#TransferID];
	        END_IF;
	        
	    END_REGION
	    
	    REGION Sensor Filter
	        
	        // FB_Sensor
	        // called as MIDB
	        
	        #TRANSFER_SENSOR(Sensor := #ReadInputSignal.TransferSensor,
	                         SensorFilterTime := #ReadTransferParameters.SensorFilterTime,
	                         FilteredSensor => #FilteredSensor);
	        
	        // front sensor filter
	        #FRONT_SENSOR_FILTER(Sensor := #FrontSensor,
	                             SensorFilterTime := #FrontSensorFilterTime);
	        
	    END_REGION
	    
	    REGION FIRE
	        
	        // Fire signal from fire system stops the whole system
	        // System can be reset from Fire status only if the fire signal is deactivated
	        
	        // FIRE ALARM ACTIVE --> STOP SYSTEM
	        IF #ReadInputSignal.FireActive THEN
	            #StopSystemFireActive := TRUE;
	        END_IF;
	        // RESET --> FIRE ALARM
	        IF #SSR.ResetSystem AND NOT #ReadInputSignal.FireActive THEN
	            #StopSystemFireActive := FALSE;
	        END_IF;
	        
	    END_REGION
	    
	END_REGION
	
	REGION Conveyor Status
	    
	    REGION Status ON
	        
	        // ----------------------------------------->>>>>>> STATUS ON <<<<<<<-----------------------------------------
	        // FB_ConveyorStatusON
	        // called as IDMB
	        
	        #TRANSFER_STATUS_ON(SystemStartActive := #SSR.StartSystem,
	                            StatusStop := #ReadTransferStatus.Stop,
	                            StatusEStop := #ReadTransferStatus.Estop,
	                            StatusManual := #ReadTransferStatus.Manual,
	                            StatusFault := #ReadTransferStatus.Fault,
	                            FireAlarmActive := #StopSystemFireActive,
	                            StatusON => #ReadTransferStatus.ON);
	        
	    END_REGION
	    
	    REGION Status Ready
	        
	        // ----------------------------------------->>>>>>> STATUS READY <<<<<<<-----------------------------------------
	        // FB_ConveyorStatusReady
	        // called as MIDB
	        
	        #TRANSFER_STATUS_READY(StatusON := #ReadTransferStatus.ON,
	                               StatusESTOP := #ReadTransferStatus.Estop,
	                               StatusFAULT := #ReadTransferStatus.Fault,
	                               StatusMAN := #ReadTransferStatus.Manual,
	                               SignalFIRE := #StopSystemFireActive,
	                               SystemAlertTime := #ReadTransferParameters.StartUpTime,
	                               StatusReady => #ReadTransferStatus.ReadytoRun);
	        
	    END_REGION
	    
	    REGION Status Occupied
	        
	        // ----------------------------------------->>>>>>> STATUS OCCUPIED <<<<<<<-----------------------------------------
	        
	        #ReadTransferStatus.Occupied :=
	        #FilteredSensor AND
	        NOT #FRONT_SENSOR_FILTER.FilteredSensor;
	        
	    END_REGION
	    
	    REGION Status Running
	        
	        // ----------------------------------------->>>>>>> STATUS RUNNING <<<<<<<-----------------------------------------
	        
	        #ReadTransferStatus.Running := #Transfer.Command_1 OR #Transfer.Command_2;
	        
	    END_REGION
	    
	    REGION Status Fault
	        
	        // Automatic reset trigger to the needed drive after wakeup from ESTOP power miss (only if needed)
	        // will trigger for every Reset active
	        
	        #AUTO_RESET(AckIN := #SSR.ResetSystem,
	                    Ack => #AutoReset);
	        
	        // ----------------------------------------->>>>>>> STATUS FAULT <<<<<<<-----------------------------------------
	        // FC_ConveyorStatusFault
	        #TRANSFER_STATUS_FAULT(FaultActive := #ReadInputSignal.Fault,
	                               ResetFault := #SSR.ResetSystem OR #AutoReset,
	                               StatusRunning := #ReadTransferStatus.Running,
	                               FaultStatus => #ReadTransferStatus.Fault);
	        
	        #ErrorReset := #SSR.ResetSystem;
	        
	    END_REGION
	    
	    REGION Status ESTOP
	        
	        // ----------------------------------------->>>>>>> STATUS ESTOP <<<<<<<-----------------------------------------
	        
	        // EMERGENCY STOP ACTIVE --> STOP SYSTEM
	        IF #ReadInputSignal.EmergencyStop THEN
	            #ReadTransferStatus.Estop := TRUE;
	        END_IF;
	        // RESET --> EMERGENCY STOP
	        IF #AutoReset AND NOT #ReadInputSignal.EmergencyStop THEN
	            #ReadTransferStatus.Estop := FALSE;
	        END_IF;
	        
	    END_REGION
	    
	    REGION Status Manual
	        
	        // ----------------------------------------->>>>>>> STATUS MANUAL <<<<<<<-----------------------------------------
	        
	        // Write to static from IO
	        // ACTIVATE --> MANUAL MODE
	        // Line A1
	        IF #Active.Line.A1 THEN
	            // SET --> MANUAL MODE
	            IF DB_Manual.Line.A1.Conveyor[#TransferID].ManualEnable THEN
	                #ReadTransferStatus.Manual := TRUE;
	            END_IF;
	            // RESET --> MANUAL MODE
	            IF NOT DB_Manual.Line.A1.Conveyor[#TransferID].ManualEnable AND #SSR.ResetSystem THEN
	                #ReadTransferStatus.Manual := FALSE;
	            END_IF;
	        END_IF;
	        // Line B1
	        IF #Active.Line.B1 THEN
	            // SET --> MANUAL MODE
	            IF DB_Manual.Line.B1.Conveyor[#TransferID].ManualEnable THEN
	                #ReadTransferStatus.Manual := TRUE;
	            END_IF;
	            // RESET --> MANUAL MODE
	            IF NOT DB_Manual.Line.B1.Conveyor[#TransferID].ManualEnable AND #SSR.ResetSystem THEN
	                #ReadTransferStatus.Manual := FALSE;
	            END_IF;
	        END_IF;
	        // Line C1
	        IF #Active.Line.C1 THEN
	            // SET --> MANUAL MODE
	            IF DB_Manual.Line.C1.Conveyor[#TransferID].ManualEnable THEN
	                #ReadTransferStatus.Manual := TRUE;
	            END_IF;
	            // RESET --> MANUAL MODE
	            IF NOT DB_Manual.Line.C1.Conveyor[#TransferID].ManualEnable AND #SSR.ResetSystem THEN
	                #ReadTransferStatus.Manual := FALSE;
	            END_IF;
	        END_IF;
	        // Line D1
	        IF #Active.Line.D1 THEN
	            // SET --> MANUAL MODE
	            IF DB_Manual.Line.D1.Conveyor[#TransferID].ManualEnable THEN
	                #ReadTransferStatus.Manual := TRUE;
	            END_IF;
	            // RESET --> MANUAL MODE
	            IF NOT DB_Manual.Line.D1.Conveyor[#TransferID].ManualEnable AND #SSR.ResetSystem THEN
	                #ReadTransferStatus.Manual := FALSE;
	            END_IF;
	        END_IF;
	        
	    END_REGION
	    
	    REGION Status Stop
	        
	        // ----------------------------------------->>>>>>> STATUS STOP <<<<<<<-----------------------------------------
	        
	        IF #SSR.StopSystem THEN
	            #ReadTransferStatus.Stop := TRUE;
	        END_IF;
	        IF #SSR.StartSystem OR #SSR.ResetSystem THEN
	            #ReadTransferStatus.Stop := FALSE;
	        END_IF;
	        
	    END_REGION
	    
	    REGION Status Blockage
	        
	        // FB_SensorBlockage
	        // called as MIDB
	        #TRANSFER_SENSOR_BLOCKAGE(IN := #ReadTransferStatus.ReadytoRun AND #FilteredSensor AND NOT #Downstream,
	                                  PT := T#15s);
	        
	        #FRONT_SENSOR_BLOCKAGE(IN := #ReadTransferStatus.ReadytoRun AND #FrontSensor AND NOT #Downstream,
	                               PT := T#15s);
	        
	        #END_SENSOR_BLOCKAGE(IN := #ReadTransferStatus.ReadytoRun AND #EndSensor AND NOT #Downstream,
	                             PT := T#15s);
	        
	        #"LEFT/RIGHT_SENSOR_BLOCKAGE"(IN := #ReadTransferStatus.ReadytoRun AND #"Left/RightSensor" AND NOT #Downstream,
	                                      PT := T#5s);
	        
	        #ReadTransferStatus.Blockage :=
	        (#TRANSFER_SENSOR_BLOCKAGE.Q OR
	        #FRONT_SENSOR_BLOCKAGE.Q OR
	        #END_SENSOR_BLOCKAGE.Q OR
	        #"LEFT/RIGHT_SENSOR_BLOCKAGE".Q) AND
	        (#TransferDirection.Straight OR
	        #TransferDirection.toRight OR
	        #TransferDirection.toLeft);
	        
	        // ==========================
	        // Sensor Blockage: HMI Alarm
	        // ==========================
	        // Sensor blockage alarm message is written to the alarm word
	        // corresponding to the active line
	        
	        REGION alarm 
	            
	            // ==========================
	            // Sensor Blockage: HMI Alarm
	            // ==========================
	            // Sensor blockage alarm message is written to the alarm word
	            // corresponding to the active line
	            // Line A1
	            IF #Active.Line.A1 THEN
	                DB_Alarm."word".Line.A1.Conveyor[#TransferID].%X0 := #ReadTransferStatus.Blockage;
	            END_IF;
	            // Line B1
	            IF #Active.Line.B1 THEN
	                DB_Alarm."word".Line.B1.Conveyor[#TransferID].%X0 := #ReadTransferStatus.Blockage;
	            END_IF;
	            // Line C1
	            IF #Active.Line.C1 THEN
	                DB_Alarm."word".Line.C1.Conveyor[#TransferID].%X0 := #ReadTransferStatus.Blockage;
	            END_IF;
	            // Line D1
	            IF #Active.Line.D1 THEN
	                DB_Alarm."word".Line.D1.Conveyor[#TransferID].%X0 := #ReadTransferStatus.Blockage;
	            END_IF;
	            
	        END_REGION
	        
	    END_REGION
	    
	    REGION Visu Color
	        
	        // each and every status of the conveyor will be mentioned by different colors in HMI panel
	        
	        #VisuColor.%X8 := #ReadTransferStatus.Blockage;
	        #VisuColor.%X0 := #ReadTransferStatus.ON;
	        #VisuColor.%X1 := #ReadTransferStatus.ReadytoRun;
	        #VisuColor.%X2 := #ReadTransferStatus.Occupied;
	        #VisuColor.%X3 := #ReadTransferStatus.Running;
	        #VisuColor.%X4 := #ReadTransferStatus.Fault;
	        #VisuColor.%X5 := #ReadTransferStatus.Estop;
	        #VisuColor.%X6 := #ReadTransferStatus.Manual;
	        #VisuColor.%X7 := #ReadTransferStatus.Stop;
	        
	        // convert word to Interger value: 
	        // color will be depends on the status priority (integer value) 
	        // reference: Conveyor image in HMI screen -> property -> Apperance   
	        
	        // Line A1
	        IF #Active.Line.A1 THEN
	            DB_VisuColor.Line.A1.Conveyor[#TransferID] :=
	            WORD_TO_INT(#VisuColor);
	        END_IF;
	        // Line B1
	        IF #Active.Line.B1 THEN
	            DB_VisuColor.Line.B1.Conveyor[#TransferID] :=
	            WORD_TO_INT(#VisuColor);
	        END_IF;
	        // Line C1
	        IF #Active.Line.C1 THEN
	            DB_VisuColor.Line.C1.Conveyor[#TransferID] :=
	            WORD_TO_INT(#VisuColor);
	        END_IF;
	        // Line D1
	        IF #Active.Line.D1 THEN
	            DB_VisuColor.Line.D1.Conveyor[#TransferID] :=
	            WORD_TO_INT(#VisuColor);
	        END_IF;
	        
	    END_REGION
	    
	    REGION Global Status
	        
